  MoveL (T7763) to (103.84, 113.06, 9.7) mm, rotated rx 180 ry 0 rz -180 deg; joints [0, 0, 0, 0, 0, 0]
  Call Extruder 0.34896
  MoveL (T7764) to (111.94, 121.16, 9.7) mm, rotated rx 180 ry 0 rz -180 deg; joints [0, 0, 0, 0, 0, 0]
  Call Extruder 0.03385
  MoveL (T7765) to (113.06, 121.16, 9.7) mm, rotated rx 180 ry 0 rz -180 deg; joints [0, 0, 0, 0, 0, 0]
  Call Extruder 0.26282
  MoveL (T7766) to (119.16, 115.06, 9.7) mm, rotated rx 180 ry 0 rz -180 deg; joints [0, 0, 0, 0, 0, 0]
  Call Extruder 0.00278
  MoveL (T7767) to (119.09, 114.99, 9.7) mm, rotated rx 180 ry 0 rz -180 deg; joints [0, 0, 0, 0, 0, 0]
  Call Extruder 0.01541
  MoveL (T7768) to (119.09, 114.48, 9.7) mm, rotated rx 180 ry 0 rz -180 deg; joints [0, 0, 0, 0, 0, 0]
  Call Extruder 0.37671
  MoveL (T7769) to (110.35, 105.74, 9.7) mm, rotated rx 180 ry 0 rz -180 deg; joints [0, 0, 0, 0, 0, 0]
  Call Extruder 0.00909
  MoveL (T7770) to (110.05, 105.74, 9.7) mm, rotated rx 180 ry 0 rz -180 deg; joints [0, 0, 0, 0, 0, 0]
  Call Extruder 0.26727
  MoveL (T7771) to (103.84, 111.94, 9.7) mm, rotated rx 180 ry 0 rz -180 deg; joints [0, 0, 0, 0, 0, 0]
  Call Extruder 0.07441
  MoveL (T7772) to (103.84, 109.5, 9.7) mm, rotated rx 180 ry 0 rz -180 deg; joints [0, 0, 0, 0, 0, 0]
  Set speed (45.0 mm/s)
  Call Extruder -1.6
  MoveL (T7773) to (103.84, 109.5, 9.7) mm, rotated rx 180 ry 0 rz -180 deg; joints [0, 0, 0, 0, 0, 0]
  Set speed (120.0 mm/s)
  MoveL (T7774) to (103.84, 109.5, 9.7) mm, rotated rx 180 ry 0 rz -180 deg; joints [0, 0, 0, 0, 0, 0]
  Call Extruder -0.38
  MoveL (T7775) to (103.84, 110.57, 9.7) mm, rotated rx 180 ry 0 rz -180 deg; joints [0, 0, 0, 0, 0, 0]
  Set speed (45.0 mm/s)
  Call Extruder -0.02
  MoveL (T7776) to (103.84, 110.57, 9.7) mm, rotated rx 180 ry 0 rz -180 deg; joints [0, 0, 0, 0, 0, 0]
  Set speed (150.0 mm/s)
  MoveL (T7777) to (103.84, 110.57, 11.7) mm, rotated rx 180 ry 0 rz -180 deg; joints [0, 0, 0, 0, 0, 0]
  MoveL (T7778) to (104.34, 103.54, 11.7) mm, rotated rx 180 ry 0 rz -180 deg; joints [0, 0, 0, 0, 0, 0]
  MoveL (T7779) to (104.34, 103.54, 9.9) mm, rotated rx 180 ry 0 rz -180 deg; joints [0, 0, 0, 0, 0, 0]
  Set speed (40.0 mm/s)
  Call Extruder 2.0
  MoveL (T7780) to (104.34, 103.54, 9.9) mm, rotated rx 180 ry 0 rz -180 deg; joints [0, 0, 0, 0, 0, 0]
  Set speed (26.4 mm/s)
  MoveL (T7781) to (104.34, 103.54, 9.9) mm, rotated rx 180 ry 0 rz -180 deg; joints [0, 0, 0, 0, 0, 0]
  Call Extruder 0.16936
  MoveL (T7782) to (109.9, 103.54, 9.9) mm, rotated rx 180 ry 0 rz -180 deg; joints [0, 0, 0, 0, 0, 0]
  Call Extruder 0.05777
  MoveL (T7783) to (109.9, 105.44, 9.9) mm, rotated rx 180 ry 0 rz -180 deg; joints [0, 0, 0, 0, 0, 0]
  Call Extruder 0.12448
  MoveL (T7784) to (113.98, 105.44, 9.9) mm, rotated rx 180 ry 0 rz -180 deg; joints [0, 0, 0, 0, 0, 0]
  Call Extruder 0.05777
  MoveL (T7785) to (113.99, 103.54, 9.9) mm, rotated rx 180 ry 0 rz -180 deg; joints [0, 0, 0, 0, 0, 0]
  Call Extruder 0.2277
  MoveL (T7786) to (121.46, 103.54, 9.9) mm, rotated rx 180 ry 0 rz -180 deg; joints [0, 0, 0, 0, 0, 0]
  Call Extruder 0.19316
  MoveL (T7787) to (121.46, 109.88, 9.9) mm, rotated rx 180 ry 0 rz -180 deg; joints [0, 0, 0, 0, 0, 0]
  Call Extruder 0.05896
  MoveL (T7788) to (119.53, 109.88, 9.9) mm, rotated rx 180 ry 0 rz -180 deg; joints [0, 0, 0, 0, 0, 0]
  Call Extruder 0.13491
  MoveL (T7789) to (119.52, 114.31, 9.9) mm, rotated rx 180 ry 0 rz -180 deg; joints [0, 0, 0, 0, 0, 0]
  Call Extruder 0.05902
  MoveL (T7790) to (121.46, 114.31, 9.9) mm, rotated rx 180 ry 0 rz -180 deg; joints [0, 0, 0, 0, 0, 0]
  Call Extruder 0.21779
  MoveL (T7791) to (121.46, 121.46, 9.9) mm, rotated rx 180 ry 0 rz -180 deg; joints [0, 0, 0, 0, 0, 0]
  Call Extruder 0.54596
  MoveL (T7792) to (103.54, 121.46, 9.9) mm, rotated rx 180 ry 0 rz -180 deg; joints [0, 0, 0, 0, 0, 0]
  Call Extruder 0.54596
  MoveL (T7793) to (103.54, 103.54, 9.9) mm, rotated rx 180 ry 0 rz -180 deg; joints [0, 0, 0, 0, 0, 0]
  Call Extruder 0.02254
  MoveL (T7794) to (104.28, 103.54, 9.9) mm, rotated rx 180 ry 0 rz -180 deg; joints [0, 0, 0, 0, 0, 0]
  Set speed (150.0 mm/s)
  MoveL (T7795) to (103.53, 103.13, 9.9) mm, rotated rx 180 ry 0 rz -180 deg; joints [0, 0, 0, 0, 0, 0]
  Set speed (26.4 mm/s)
  MoveL (T7796) to (103.53, 103.13, 9.9) mm, rotated rx 180 ry 0 rz -180 deg; joints [0, 0, 0, 0, 0, 0]
  Call Extruder 0.20634
  MoveL (T7797) to (110.31, 103.13, 9.9) mm, rotated rx 180 ry 0 rz -180 deg; joints [0, 0, 0, 0, 0, 0]
  Call Extruder 0.05777
  MoveL (T7798) to (110.31, 105.03, 9.9) mm, rotated rx 180 ry 0 rz -180 deg; joints [0, 0, 0, 0, 0, 0]
  Call Extruder 0.09969
  MoveL (T7799) to (113.58, 105.03, 9.9) mm, rotated rx 180 ry 0 rz -180 deg; joints [0, 0, 0, 0, 0, 0]
  Call Extruder 0.05777
  MoveL (T7800) to (113.58, 103.13, 9.9) mm, rotated rx 180 ry 0 rz -180 deg; joints [0, 0, 0, 0, 0, 0]
  Call Extruder 0.2525
  MoveL (T7801) to (121.87, 103.13, 9.9) mm, rotated rx 180 ry 0 rz -180 deg; joints [0, 0, 0, 0, 0, 0]
  Call Extruder 0.21796
  MoveL (T7802) to (121.87, 110.29, 9.9) mm, rotated rx 180 ry 0 rz -180 deg; joints [0, 0, 0, 0, 0, 0]
  Call Extruder 0.05897
  MoveL (T7803) to (119.93, 110.29, 9.9) mm, rotated rx 180 ry 0 rz -180 deg; joints [0, 0, 0, 0, 0, 0]
  Call Extruder 0.11013
  MoveL (T7804) to (119.93, 113.9, 9.9) mm, rotated rx 180 ry 0 rz -180 deg; joints [0, 0, 0, 0, 0, 0]
  Call Extruder 0.05902
  MoveL (T7805) to (121.87, 113.91, 9.9) mm, rotated rx 180 ry 0 rz -180 deg; joints [0, 0, 0, 0, 0, 0]
  Call Extruder 0.24258
  MoveL (T7806) to (121.87, 121.87, 9.9) mm, rotated rx 180 ry 0 rz -180 deg; joints [0, 0, 0, 0, 0, 0]
  Call Extruder 0.57077
  MoveL (T7807) to (103.13, 121.87, 9.9) mm, rotated rx 180 ry 0 rz -180 deg; joints [0, 0, 0, 0, 0, 0]
  Call Extruder 0.57077
  MoveL (T7808) to (103.13, 103.13, 9.9) mm, rotated rx 180 ry 0 rz -180 deg; joints [0, 0, 0, 0, 0, 0]
  Call Extruder 0.01036
  MoveL (T7809) to (103.47, 103.13, 9.9) mm, rotated rx 180 ry 0 rz -180 deg; joints [0, 0, 0, 0, 0, 0]
  Set speed (150.0 mm/s)
  MoveL (T7810) to (102.72, 102.81, 9.9) mm, rotated rx 180 ry 0 rz -180 deg; joints [0, 0, 0, 0, 0, 0]
  Set speed (25.0 mm/s)
  MoveL (T7811) to (102.72, 102.81, 9.9) mm, rotated rx 180 ry 0 rz -180 deg; joints [0, 0, 0, 0, 0, 0]
  Call Extruder 0.00259
  MoveL (T7812) to (102.72, 102.72, 9.9) mm, rotated rx 180 ry 0 rz -180 deg; joints [0, 0, 0, 0, 0, 0]
  Call Extruder 0.24332
  MoveL (T7813) to (110.71, 102.72, 9.9) mm, rotated rx 180 ry 0 rz -180 deg; joints [0, 0, 0, 0, 0, 0]
  Call Extruder 0.05777
  MoveL (T7814) to (110.71, 104.62, 9.9) mm, rotated rx 180 ry 0 rz -180 deg; joints [0, 0, 0, 0, 0, 0]
  Call Extruder 0.0749
  MoveL (T7815) to (113.17, 104.62, 9.9) mm, rotated rx 180 ry 0 rz -180 deg; joints [0, 0, 0, 0, 0, 0]
  Call Extruder 0.05777
  MoveL (T7816) to (113.17, 102.72, 9.9) mm, rotated rx 180 ry 0 rz -180 deg; joints [0, 0, 0, 0, 0, 0]
  Call Extruder 0.27729
  MoveL (T7817) to (122.28, 102.72, 9.9) mm, rotated rx 180 ry 0 rz -180 deg; joints [0, 0, 0, 0, 0, 0]
  Call Extruder 0.24275
  MoveL (T7818) to (122.28, 110.69, 9.9) mm, rotated rx 180 ry 0 rz -180 deg; joints [0, 0, 0, 0, 0, 0]
  Call Extruder 0.05897
  MoveL (T7819) to (120.34, 110.69, 9.9) mm, rotated rx 180 ry 0 rz -180 deg; joints [0, 0, 0, 0, 0, 0]
  Call Extruder 0.08535
  MoveL (T7820) to (120.34, 113.5, 9.9) mm, rotated rx 180 ry 0 rz -180 deg; joints [0, 0, 0, 0, 0, 0]
  Call Extruder 0.05901
  MoveL (T7821) to (122.28, 113.5, 9.9) mm, rotated rx 180 ry 0 rz -180 deg; joints [0, 0, 0, 0, 0, 0]
  Call Extruder 0.26736
  MoveL (T7822) to (122.28, 122.28, 9.9) mm, rotated rx 180 ry 0 rz -180 deg; joints [0, 0, 0, 0, 0, 0]
  Call Extruder 0.59557
  MoveL (T7823) to (102.72, 122.28, 9.9) mm, rotated rx 180 ry 0 rz -180 deg; joints [0, 0, 0, 0, 0, 0]
  Call Extruder 0.59115
  MoveL (T7824) to (102.72, 102.87, 9.9) mm, rotated rx 180 ry 0 rz -180 deg; joints [0, 0, 0, 0, 0, 0]
  Set speed (150.0 mm/s)
  MoveL (T7825) to (102.78, 102.75, 9.9) mm, rotated rx 180 ry 0 rz -180 deg; joints [0, 0, 0, 0, 0, 0]
  Set speed (45.0 mm/s)
  Call Extruder -1.6
  MoveL (T7826) to (102.78, 102.75, 9.9) mm, rotated rx 180 ry 0 rz -180 deg; joints [0, 0, 0, 0, 0, 0]
  Set speed (120.0 mm/s)
  MoveL (T7827) to (102.78, 102.75, 9.9) mm, rotated rx 180 ry 0 rz -180 deg; joints [0, 0, 0, 0, 0, 0]
  Call Extruder -0.05166
  MoveL (T7828) to (102.72, 102.72, 9.9) mm, rotated rx 180 ry 0 rz -180 deg; joints [0, 0, 0, 0, 0, 0]
  Call Extruder -0.32834
  MoveL (T7829) to (103.65, 102.72, 9.9) mm, rotated rx 180 ry 0 rz -180 deg; joints [0, 0, 0, 0, 0, 0]
  Set speed (45.0 mm/s)
  Call Extruder -0.02
  MoveL (T7830) to (103.65, 102.72, 9.9) mm, rotated rx 180 ry 0 rz -180 deg; joints [0, 0, 0, 0, 0, 0]
  Set speed (150.0 mm/s)
  MoveL (T7831) to (103.65, 102.72, 11.9) mm, rotated rx 180 ry 0 rz -180 deg; joints [0, 0, 0, 0, 0, 0]
  MoveL (T7832) to (106.29, 103.84, 11.9) mm, rotated rx 180 ry 0 rz -180 deg; joints [0, 0, 0, 0, 0, 0]
  MoveL (T7833) to (106.29, 103.84, 9.9) mm, rotated rx 180 ry 0 rz -180 deg; joints [0, 0, 0, 0, 0, 0]
  Set speed (40.0 mm/s)
  Call Extruder 2.0
  MoveL (T7834) to (106.29, 103.84, 9.9) mm, rotated rx 180 ry 0 rz -180 deg; joints [0, 0, 0, 0, 0, 0]
  Set speed (26.4 mm/s)
  MoveL (T7835) to (106.29, 103.84, 9.9) mm, rotated rx 180 ry 0 rz -180 deg; joints [0, 0, 0, 0, 0, 0]
  Call Extruder 0.07441
  MoveL (T7836) to (103.84, 103.84, 9.9) mm, rotated rx 180 ry 0 rz -180 deg; joints [0, 0, 0, 0, 0, 0]
  Call Extruder 0.7458
  MoveL (T7837) to (121.16, 121.16, 9.9) mm, rotated rx 180 ry 0 rz -180 deg; joints [0, 0, 0, 0, 0, 0]
  Call Extruder 0.07441
  MoveL (T7838) to (118.71, 121.16, 9.9) mm, rotated rx 180 ry 0 rz -180 deg; joints [0, 0, 0, 0, 0, 0]
  Set speed (45.0 mm/s)
  Call Extruder -1.6
  MoveL (T7839) to (118.71, 121.16, 9.9) mm, rotated rx 180 ry 0 rz -180 deg; joints [0, 0, 0, 0, 0, 0]
  Set speed (120.0 mm/s)
  MoveL (T7840) to (118.71, 121.16, 9.9) mm, rotated rx 180 ry 0 rz -180 deg; joints [0, 0, 0, 0, 0, 0]
  Call Extruder -0.38
  MoveL (T7841) to (119.78, 121.16, 9.9) mm, rotated rx 180 ry 0 rz -180 deg; joints [0, 0, 0, 0, 0, 0]
  Set speed (45.0 mm/s)
  Call Extruder -0.02
  MoveL (T7842) to (119.78, 121.16, 9.9) mm, rotated rx 180 ry 0 rz -180 deg; joints [0, 0, 0, 0, 0, 0]
  Set speed (150.0 mm/s)
  MoveL (T7843) to (119.78, 121.16, 11.9) mm, rotated rx 180 ry 0 rz -180 deg; joints [0, 0, 0, 0, 0, 0]
  MoveL (T7844) to (121.16, 116.35, 11.9) mm, rotated rx 180 ry 0 rz -180 deg; joints [0, 0, 0, 0, 0, 0]
  MoveL (T7845) to (121.16, 116.35, 9.9) mm, rotated rx 180 ry 0 rz -180 deg; joints [0, 0, 0, 0, 0, 0]
  Set speed (40.0 mm/s)
  Call Extruder 2.0
  MoveL (T7846) to (121.16, 116.35, 9.9) mm, rotated rx 180 ry 0 rz -180 deg; joints [0, 0, 0, 0, 0, 0]
  Set speed (26.4 mm/s)
  MoveL (T7847) to (121.16, 116.35, 9.9) mm, rotated rx 180 ry 0 rz -180 deg; joints [0, 0, 0, 0, 0, 0]
  Call Extruder 0.02808
  MoveL (T7848) to (121.16, 115.42, 9.9) mm, rotated rx 180 ry 0 rz -180 deg; joints [0, 0, 0, 0, 0, 0]
  Call Extruder 0.03432
  MoveL (T7849) to (120.03, 115.42, 9.9) mm, rotated rx 180 ry 0 rz -180 deg; joints [0, 0, 0, 0, 0, 0]
  Call Extruder 0.04854
  MoveL (T7850) to (121.16, 116.55, 9.9) mm, rotated rx 180 ry 0 rz -180 deg; joints [0, 0, 0, 0, 0, 0]
  Call Extruder 0.03385
  MoveL (T7851) to (121.16, 117.66, 9.9) mm, rotated rx 180 ry 0 rz -180 deg; joints [0, 0, 0, 0, 0, 0]
  Call Extruder 0.15054
  MoveL (T7852) to (117.66, 121.16, 9.9) mm, rotated rx 180 ry 0 rz -180 deg; joints [0, 0, 0, 0, 0, 0]
  Call Extruder 0.03385
  MoveL (T7853) to (116.55, 121.16, 9.9) mm, rotated rx 180 ry 0 rz -180 deg; joints [0, 0, 0, 0, 0, 0]
  Call Extruder 0.54738
  MoveL (T7854) to (103.84, 108.45, 9.9) mm, rotated rx 180 ry 0 rz -180 deg; joints [0, 0, 0, 0, 0, 0]
  Call Extruder 0.03385
  MoveL (T7855) to (103.84, 107.34, 9.9) mm, rotated rx 180 ry 0 rz -180 deg; joints [0, 0, 0, 0, 0, 0]
  Call Extruder 0.15054
  MoveL (T7856) to (107.34, 103.84, 9.9) mm, rotated rx 180 ry 0 rz -180 deg; joints [0, 0, 0, 0, 0, 0]
  Call Extruder 0.03385
  MoveL (T7857) to (108.45, 103.84, 9.9) mm, rotated rx 180 ry 0 rz -180 deg; joints [0, 0, 0, 0, 0, 0]
  Call Extruder 0.02461
  MoveL (T7858) to (109.02, 104.42, 9.9) mm, rotated rx 180 ry 0 rz -180 deg; joints [0, 0, 0, 0, 0, 0]
  Call Extruder 0.03458
  MoveL (T7859) to (109.02, 105.55, 9.9) mm, rotated rx 180 ry 0 rz -180 deg; joints [0, 0, 0, 0, 0, 0]
  Call Extruder 0.01376
  MoveL (T7860) to (109.34, 105.87, 9.9) mm, rotated rx 180 ry 0 rz -180 deg; joints [0, 0, 0, 0, 0, 0]
  Call Extruder 0.01427
  MoveL (T7861) to (109.81, 105.87, 9.9) mm, rotated rx 180 ry 0 rz -180 deg; joints [0, 0, 0, 0, 0, 0]
  Call Extruder 0.00269
  MoveL (T7862) to (109.87, 105.81, 9.9) mm, rotated rx 180 ry 0 rz -180 deg; joints [0, 0, 0, 0, 0, 0]
  Set speed (150.0 mm/s)
  MoveL (T7863) to (109.78, 104.52, 9.9) mm, rotated rx 180 ry 0 rz -180 deg; joints [0, 0, 0, 0, 0, 0]
  Set speed (26.4 mm/s)
  MoveL (T7864) to (109.78, 104.52, 9.9) mm, rotated rx 180 ry 0 rz -180 deg; joints [0, 0, 0, 0, 0, 0]
  Call Extruder 0.01563
  MoveL (T7865) to (109.43, 104.17, 9.9) mm, rotated rx 180 ry 0 rz -180 deg; joints [0, 0, 0, 0, 0, 0]
  Call Extruder 0.01901
  MoveL (T7866) to (109.43, 104.77, 9.9) mm, rotated rx 180 ry 0 rz -180 deg; joints [0, 0, 0, 0, 0, 0]
  Call Extruder 0.00741
  MoveL (T7867) to (109.59, 104.94, 9.9) mm, rotated rx 180 ry 0 rz -180 deg; joints [0, 0, 0, 0, 0, 0]
  Call Extruder 0.01671
  MoveL (T7868) to (109.59, 105.46, 9.9) mm, rotated rx 180 ry 0 rz -180 deg; joints [0, 0, 0, 0, 0, 0]
  Call Extruder 0.0023
  MoveL (T7869) to (109.52, 105.46, 9.9) mm, rotated rx 180 ry 0 rz -180 deg; joints [0, 0, 0, 0, 0, 0]
  Call Extruder 0.01238
  MoveL (T7870) to (109.25, 105.19, 9.9) mm, rotated rx 180 ry 0 rz -180 deg; joints [0, 0, 0, 0, 0, 0]
  Set speed (45.0 mm/s)
  Call Extruder -1.6
  MoveL (T7871) to (109.25, 105.19, 9.9) mm, rotated rx 180 ry 0 rz -180 deg; joints [0, 0, 0, 0, 0, 0]
  Set speed (120.0 mm/s)
  MoveL (T7872) to (109.25, 105.19, 9.9) mm, rotated rx 180 ry 0 rz -180 deg; joints [0, 0, 0, 0, 0, 0]
  Call Extruder -0.13905
  MoveL (T7873) to (109.52, 105.46, 9.9) mm, rotated rx 180 ry 0 rz -180 deg; joints [0, 0, 0, 0, 0, 0]
  Call Extruder -0.02586
  MoveL (T7874) to (109.59, 105.46, 9.9) mm, rotated rx 180 ry 0 rz -180 deg; joints [0, 0, 0, 0, 0, 0]
  Call Extruder -0.18771
  MoveL (T7875) to (109.59, 104.94, 9.9) mm, rotated rx 180 ry 0 rz -180 deg; joints [0, 0, 0, 0, 0, 0]
  Call Extruder -0.02738
  MoveL (T7876) to (109.54, 104.88, 9.9) mm, rotated rx 180 ry 0 rz -180 deg; joints [0, 0, 0, 0, 0, 0]
  Set speed (45.0 mm/s)
  Call Extruder -0.02
  MoveL (T7877) to (109.54, 104.88, 9.9) mm, rotated rx 180 ry 0 rz -180 deg; joints [0, 0, 0, 0, 0, 0]
  Set speed (150.0 mm/s)
  MoveL (T7878) to (109.54, 104.88, 11.9) mm, rotated rx 180 ry 0 rz -180 deg; joints [0, 0, 0, 0, 0, 0]
  MoveL (T7879) to (112.14, 105.74, 11.9) mm, rotated rx 180 ry 0 rz -180 deg; joints [0, 0, 0, 0, 0, 0]
  MoveL (T7880) to (112.14, 105.74, 9.9) mm, rotated rx 180 ry 0 rz -180 deg; joints [0, 0, 0, 0, 0, 0]
  Set speed (40.0 mm/s)
  Call Extruder 2.0
  MoveL (T7881) to (112.14, 105.74, 9.9) mm, rotated rx 180 ry 0 rz -180 deg; joints [0, 0, 0, 0, 0, 0]
  Set speed (26.4 mm/s)
  MoveL (T7882) to (112.14, 105.74, 9.9) mm, rotated rx 180 ry 0 rz -180 deg; joints [0, 0, 0, 0, 0, 0]
  Call Extruder 0.05515
  MoveL (T7883) to (113.95, 105.74, 9.9) mm, rotated rx 180 ry 0 rz -180 deg; joints [0, 0, 0, 0, 0, 0]
  Call Extruder 0.00557
  MoveL (T7884) to (114.08, 105.87, 9.9) mm, rotated rx 180 ry 0 rz -180 deg; joints [0, 0, 0, 0, 0, 0]
  Call Extruder 0.01369
  MoveL (T7885) to (114.52, 105.87, 9.9) mm, rotated rx 180 ry 0 rz -180 deg; joints [0, 0, 0, 0, 0, 0]
  Call Extruder 0.46011
  MoveL (T7886) to (103.84, 116.55, 9.9) mm, rotated rx 180 ry 0 rz -180 deg; joints [0, 0, 0, 0, 0, 0]
  Call Extruder 0.03385
  MoveL (T7887) to (103.84, 117.66, 9.9) mm, rotated rx 180 ry 0 rz -180 deg; joints [0, 0, 0, 0, 0, 0]
  Call Extruder 0.15054
  MoveL (T7888) to (107.34, 121.16, 9.9) mm, rotated rx 180 ry 0 rz -180 deg; joints [0, 0, 0, 0, 0, 0]
  Call Extruder 0.03385
  MoveL (T7889) to (108.45, 121.16, 9.9) mm, rotated rx 180 ry 0 rz -180 deg; joints [0, 0, 0, 0, 0, 0]
  Call Extruder 0.46399
  MoveL (T7890) to (119.22, 110.39, 9.9) mm, rotated rx 180 ry 0 rz -180 deg; joints [0, 0, 0, 0, 0, 0]
  Call Extruder 0.01148
  MoveL (T7891) to (119.22, 110.01, 9.9) mm, rotated rx 180 ry 0 rz -180 deg; joints [0, 0, 0, 0, 0, 0]
  Call Extruder 0.18856
  MoveL (T7892) to (114.84, 105.63, 9.9) mm, rotated rx 180 ry 0 rz -180 deg; joints [0, 0, 0, 0, 0, 0]
  Call Extruder 0.00351
  MoveL (T7893) to (114.92, 105.55, 9.9) mm, rotated rx 180 ry 0 rz -180 deg; joints [0, 0, 0, 0, 0, 0]
  Call Extruder 0.00247
  MoveL (T7894) to (114.92, 105.47, 9.9) mm, rotated rx 180 ry 0 rz -180 deg; joints [0, 0, 0, 0, 0, 0]
  Call Extruder 0.07002
  MoveL (T7895) to (116.55, 103.84, 9.9) mm, rotated rx 180 ry 0 rz -180 deg; joints [0, 0, 0, 0, 0, 0]
  Call Extruder 0.03385
  MoveL (T7896) to (117.66, 103.84, 9.9) mm, rotated rx 180 ry 0 rz -180 deg; joints [0, 0, 0, 0, 0, 0]
  Call Extruder 0.15054
  MoveL (T7897) to (121.16, 107.34, 9.9) mm, rotated rx 180 ry 0 rz -180 deg; joints [0, 0, 0, 0, 0, 0]
  Call Extruder 0.03385
  MoveL (T7898) to (121.16, 108.45, 9.9) mm, rotated rx 180 ry 0 rz -180 deg; joints [0, 0, 0, 0, 0, 0]
  Call Extruder 0.01201
  MoveL (T7899) to (120.88, 108.73, 9.9) mm, rotated rx 180 ry 0 rz -180 deg; joints [0, 0, 0, 0, 0, 0]
  Call Extruder 0.04458
  MoveL (T7900) to (119.41, 108.73, 9.9) mm, rotated rx 180 ry 0 rz -180 deg; joints [0, 0, 0, 0, 0, 0]
  Call Extruder 0.01373
  MoveL (T7901) to (119.09, 109.05, 9.9) mm, rotated rx 180 ry 0 rz -180 deg; joints [0, 0, 0, 0, 0, 0]
  Call Extruder 0.01609
  MoveL (T7902) to (119.09, 109.58, 9.9) mm, rotated rx 180 ry 0 rz -180 deg; joints [0, 0, 0, 0, 0, 0]
  Set speed (45.0 mm/s)
  Call Extruder -1.6
  MoveL (T7903) to (119.09, 109.58, 9.9) mm, rotated rx 180 ry 0 rz -180 deg; joints [0, 0, 0, 0, 0, 0]
  Set speed (120.0 mm/s)
  MoveL (T7904) to (119.09, 109.58, 9.9) mm, rotated rx 180 ry 0 rz -180 deg; joints [0, 0, 0, 0, 0, 0]
  Call Extruder -0.18818
  MoveL (T7905) to (119.09, 109.05, 9.9) mm, rotated rx 180 ry 0 rz -180 deg; joints [0, 0, 0, 0, 0, 0]
  Call Extruder -0.16059
  MoveL (T7906) to (119.41, 108.73, 9.9) mm, rotated rx 180 ry 0 rz -180 deg; joints [0, 0, 0, 0, 0, 0]
  Call Extruder -0.03122
  MoveL (T7907) to (119.5, 108.73, 9.9) mm, rotated rx 180 ry 0 rz -180 deg; joints [0, 0, 0, 0, 0, 0]
  Set speed (45.0 mm/s)
  Call Extruder -0.02
  MoveL (T7908) to (119.5, 108.73, 9.9) mm, rotated rx 180 ry 0 rz -180 deg; joints [0, 0, 0, 0, 0, 0]
  Set speed (150.0 mm/s)
  MoveL (T7909) to (119.5, 108.73, 11.9) mm, rotated rx 180 ry 0 rz -180 deg; joints [0, 0, 0, 0, 0, 0]
  MoveL (T7910) to (121.34, 109.33, 11.9) mm, rotated rx 180 ry 0 rz -180 deg; joints [0, 0, 0, 0, 0, 0]
  MoveL (T7911) to (121.34, 109.33, 9.9) mm, rotated rx 180 ry 0 rz -180 deg; joints [0, 0, 0, 0, 0, 0]
  Set speed (40.0 mm/s)
  Call Extruder 2.0
  MoveL (T7912) to (121.34, 109.33, 9.9) mm, rotated rx 180 ry 0 rz -180 deg; joints [0, 0, 0, 0, 0, 0]
  Set speed (26.4 mm/s)
  MoveL (T7913) to (121.34, 109.33, 9.9) mm, rotated rx 180 ry 0 rz -180 deg; joints [0, 0, 0, 0, 0, 0]
  Call Extruder 0.01001
  MoveL (T7914) to (121.14, 109.14, 9.9) mm, rotated rx 180 ry 0 rz -180 deg; joints [0, 0, 0, 0, 0, 0]
  Call Extruder 0.02524
  MoveL (T7915) to (120.45, 109.14, 9.9) mm, rotated rx 180 ry 0 rz -180 deg; joints [0, 0, 0, 0, 0, 0]
  Call Extruder 0.02268
  MoveL (T7916) to (120.89, 109.58, 9.9) mm, rotated rx 180 ry 0 rz -180 deg; joints [0, 0, 0, 0, 0, 0]
  Call Extruder 0.02524
  MoveL (T7917) to (120.2, 109.58, 9.9) mm, rotated rx 180 ry 0 rz -180 deg; joints [0, 0, 0, 0, 0, 0]
  Call Extruder 0.02268
  MoveL (T7918) to (119.76, 109.14, 9.9) mm, rotated rx 180 ry 0 rz -180 deg; joints [0, 0, 0, 0, 0, 0]
  Call Extruder 0.00667
  MoveL (T7919) to (119.58, 109.14, 9.9) mm, rotated rx 180 ry 0 rz -180 deg; joints [0, 0, 0, 0, 0, 0]
  Call Extruder 0.00418
  MoveL (T7920) to (119.5, 109.22, 9.9) mm, rotated rx 180 ry 0 rz -180 deg; joints [0, 0, 0, 0, 0, 0]
  Call Extruder 0.01263
  MoveL (T7921) to (119.5, 109.56, 9.9) mm, rotated rx 180 ry 0 rz -180 deg; joints [0, 0, 0, 0, 0, 0]
  Call Extruder 0.01011
  MoveL (T7922) to (119.69, 109.76, 9.9) mm, rotated rx 180 ry 0 rz -180 deg; joints [0, 0, 0, 0, 0, 0]
  Set speed (45.0 mm/s)
  Call Extruder -1.6
  MoveL (T7923) to (119.69, 109.76, 9.9) mm, rotated rx 180 ry 0 rz -180 deg; joints [0, 0, 0, 0, 0, 0]
  Set speed (120.0 mm/s)
  MoveL (T7924) to (119.69, 109.76, 9.9) mm, rotated rx 180 ry 0 rz -180 deg; joints [0, 0, 0, 0, 0, 0]
  Call Extruder -0.09855
  MoveL (T7925) to (119.5, 109.56, 9.9) mm, rotated rx 180 ry 0 rz -180 deg; joints [0, 0, 0, 0, 0, 0]
  Call Extruder -0.1231
  MoveL (T7926) to (119.5, 109.22, 9.9) mm, rotated rx 180 ry 0 rz -180 deg; joints [0, 0, 0, 0, 0, 0]
  Call Extruder -0.04075
  MoveL (T7927) to (119.58, 109.14, 9.9) mm, rotated rx 180 ry 0 rz -180 deg; joints [0, 0, 0, 0, 0, 0]
  Call Extruder -0.06497
  MoveL (T7928) to (119.76, 109.14, 9.9) mm, rotated rx 180 ry 0 rz -180 deg; joints [0, 0, 0, 0, 0, 0]
  Call Extruder -0.05262
  MoveL (T7929) to (119.87, 109.24, 9.9) mm, rotated rx 180 ry 0 rz -180 deg; joints [0, 0, 0, 0, 0, 0]
  Set speed (45.0 mm/s)
  Call Extruder -0.02
  MoveL (T7930) to (119.87, 109.24, 9.9) mm, rotated rx 180 ry 0 rz -180 deg; joints [0, 0, 0, 0, 0, 0]
  Set speed (150.0 mm/s)
  MoveL (T7931) to (119.87, 109.24, 11.9) mm, rotated rx 180 ry 0 rz -180 deg; joints [0, 0, 0, 0, 0, 0]
  MoveL (T7932) to (121.14, 115.2, 11.9) mm, rotated rx 180 ry 0 rz -180 deg; joints [0, 0, 0, 0, 0, 0]
  MoveL (T7933) to (121.14, 115.2, 9.9) mm, rotated rx 180 ry 0 rz -180 deg; joints [0, 0, 0, 0, 0, 0]
  Set speed (40.0 mm/s)
  Call Extruder 2.0
  MoveL (T7934) to (121.14, 115.2, 9.9) mm, rotated rx 180 ry 0 rz -180 deg; joints [0, 0, 0, 0, 0, 0]
  Set speed (26.4 mm/s)
  MoveL (T7935) to (121.14, 115.2, 9.9) mm, rotated rx 180 ry 0 rz -180 deg; joints [0, 0, 0, 0, 0, 0]
  Call Extruder 0.02922
  MoveL (T7936) to (120.56, 114.62, 9.9) mm, rotated rx 180 ry 0 rz -180 deg; joints [0, 0, 0, 0, 0, 0]
  Call Extruder 0.02361
  MoveL (T7937) to (119.89, 114.61, 9.9) mm, rotated rx 180 ry 0 rz -180 deg; joints [0, 0, 0, 0, 0, 0]
  Call Extruder 0.02006
  MoveL (T7938) to (120.29, 115.02, 9.9) mm, rotated rx 180 ry 0 rz -180 deg; joints [0, 0, 0, 0, 0, 0]
  Call Extruder 0.02361
  MoveL (T7939) to (119.62, 115.02, 9.9) mm, rotated rx 180 ry 0 rz -180 deg; joints [0, 0, 0, 0, 0, 0]
  Call Extruder 0.0155
  MoveL (T7940) to (119.31, 114.7, 9.9) mm, rotated rx 180 ry 0 rz -180 deg; joints [0, 0, 0, 0, 0, 0]
  Set speed (45.0 mm/s)
  Call Extruder -1.6
  MoveL (T7941) to (119.31, 114.7, 9.9) mm, rotated rx 180 ry 0 rz -180 deg; joints [0, 0, 0, 0, 0, 0]
  Set speed (120.0 mm/s)
  MoveL (T7942) to (119.31, 114.7, 9.9) mm, rotated rx 180 ry 0 rz -180 deg; joints [0, 0, 0, 0, 0, 0]
  Call Extruder -0.15638
  MoveL (T7943) to (119.62, 115.02, 9.9) mm, rotated rx 180 ry 0 rz -180 deg; joints [0, 0, 0, 0, 0, 0]
  Call Extruder -0.22362
  MoveL (T7944) to (120.25, 115.02, 9.9) mm, rotated rx 180 ry 0 rz -180 deg; joints [0, 0, 0, 0, 0, 0]
  Set speed (45.0 mm/s)
  Call Extruder -0.02
  MoveL (T7945) to (120.25, 115.02, 9.9) mm, rotated rx 180 ry 0 rz -180 deg; joints [0, 0, 0, 0, 0, 0]
  Set speed (150.0 mm/s)
  MoveL (T7946) to (120.25, 115.02, 11.9) mm, rotated rx 180 ry 0 rz -180 deg; joints [0, 0, 0, 0, 0, 0]
  MoveL (T7947) to (118.71, 103.84, 11.9) mm, rotated rx 180 ry 0 rz -180 deg; joints [0, 0, 0, 0, 0, 0]
  MoveL (T7948) to (118.71, 103.84, 9.9) mm, rotated rx 180 ry 0 rz -180 deg; joints [0, 0, 0, 0, 0, 0]
  Set speed (40.0 mm/s)
  Call Extruder 2.0
  MoveL (T7949) to (118.71, 103.84, 9.9) mm, rotated rx 180 ry 0 rz -180 deg; joints [0, 0, 0, 0, 0, 0]
  Set speed (26.4 mm/s)
  MoveL (T7950) to (118.71, 103.84, 9.9) mm, rotated rx 180 ry 0 rz -180 deg; joints [0, 0, 0, 0, 0, 0]
  Call Extruder 0.07441
  MoveL (T7951) to (121.16, 103.84, 9.9) mm, rotated rx 180 ry 0 rz -180 deg; joints [0, 0, 0, 0, 0, 0]
  Call Extruder 0.7458
  MoveL (T7952) to (103.84, 121.16, 9.9) mm, rotated rx 180 ry 0 rz -180 deg; joints [0, 0, 0, 0, 0, 0]
  Call Extruder 0.07441
  MoveL (T7953) to (106.29, 121.16, 9.9) mm, rotated rx 180 ry 0 rz -180 deg; joints [0, 0, 0, 0, 0, 0]
  Set speed (45.0 mm/s)
  Call Extruder -1.6
  MoveL (T7954) to (106.29, 121.16, 9.9) mm, rotated rx 180 ry 0 rz -180 deg; joints [0, 0, 0, 0, 0, 0]
  Set speed (120.0 mm/s)
  MoveL (T7955) to (106.29, 121.16, 9.9) mm, rotated rx 180 ry 0 rz -180 deg; joints [0, 0, 0, 0, 0, 0]
  Call Extruder -0.38
  MoveL (T7956) to (105.22, 121.16, 9.9) mm, rotated rx 180 ry 0 rz -180 deg; joints [0, 0, 0, 0, 0, 0]
  Set speed (45.0 mm/s)
  Call Extruder -0.02
  MoveL (T7957) to (105.22, 121.16, 9.9) mm, rotated rx 180 ry 0 rz -180 deg; joints [0, 0, 0, 0, 0, 0]
  Set speed (150.0 mm/s)
  MoveL (T7958) to (105.22, 121.16, 11.9) mm, rotated rx 180 ry 0 rz -180 deg; joints [0, 0, 0, 0, 0, 0]
  MoveL (T7959) to (103.84, 115.5, 11.9) mm, rotated rx 180 ry 0 rz -180 deg; joints [0, 0, 0, 0, 0, 0]
  MoveL (T7960) to (103.84, 115.5, 9.9) mm, rotated rx 180 ry 0 rz -180 deg; joints [0, 0, 0, 0, 0, 0]
  Set speed (40.0 mm/s)
  Call Extruder 2.0
  MoveL (T7961) to (103.84, 115.5, 9.9) mm, rotated rx 180 ry 0 rz -180 deg; joints [0, 0, 0, 0, 0, 0]
  Set speed (26.4 mm/s)
  MoveL (T7962) to (103.84, 115.5, 9.9) mm, rotated rx 180 ry 0 rz -180 deg; joints [0, 0, 0, 0, 0, 0]
  Call Extruder 0.07441
  MoveL (T7963) to (103.84, 113.06, 9.9) mm, rotated rx 180 ry 0 rz -180 deg; joints [0, 0, 0, 0, 0, 0]
  Call Extruder 0.34896
  MoveL (T7964) to (111.94, 121.16, 9.9) mm, rotated rx 180 ry 0 rz -180 deg; joints [0, 0, 0, 0, 0, 0]
  Call Extruder 0.03385
  MoveL (T7965) to (113.06, 121.16, 9.9) mm, rotated rx 180 ry 0 rz -180 deg; joints [0, 0, 0, 0, 0, 0]
  Call Extruder 0.26038
  MoveL (T7966) to (119.1, 115.11, 9.9) mm, rotated rx 180 ry 0 rz -180 deg; joints [0, 0, 0, 0, 0, 0]
  Call Extruder 0.0191
  MoveL (T7967) to (119.09, 114.48, 9.9) mm, rotated rx 180 ry 0 rz -180 deg; joints [0, 0, 0, 0, 0, 0]
  Call Extruder 0.37671
  MoveL (T7968) to (110.35, 105.74, 9.9) mm, rotated rx 180 ry 0 rz -180 deg; joints [0, 0, 0, 0, 0, 0]
  Call Extruder 0.0091
  MoveL (T7969) to (110.05, 105.74, 9.9) mm, rotated rx 180 ry 0 rz -180 deg; joints [0, 0, 0, 0, 0, 0]
  Call Extruder 0.26726
  MoveL (T7970) to (103.84, 111.94, 9.9) mm, rotated rx 180 ry 0 rz -180 deg; joints [0, 0, 0, 0, 0, 0]
  Call Extruder 0.07441
  MoveL (T7971) to (103.84, 109.5, 9.9) mm, rotated rx 180 ry 0 rz -180 deg; joints [0, 0, 0, 0, 0, 0]
  Set speed (45.0 mm/s)
  Call Extruder -1.6
  MoveL (T7972) to (103.84, 109.5, 9.9) mm, rotated rx 180 ry 0 rz -180 deg; joints [0, 0, 0, 0, 0, 0]
  Set speed (120.0 mm/s)
  MoveL (T7973) to (103.84, 109.5, 9.9) mm, rotated rx 180 ry 0 rz -180 deg; joints [0, 0, 0, 0, 0, 0]
  Call Extruder -0.38
  MoveL (T7974) to (103.84, 110.57, 9.9) mm, rotated rx 180 ry 0 rz -180 deg; joints [0, 0, 0, 0, 0, 0]
  Set speed (45.0 mm/s)
  Call Extruder -0.02
  MoveL (T7975) to (103.84, 110.57, 9.9) mm, rotated rx 180 ry 0 rz -180 deg; joints [0, 0, 0, 0, 0, 0]
  Set speed (150.0 mm/s)
  MoveL (T7976) to (103.84, 110.57, 11.9) mm, rotated rx 180 ry 0 rz -180 deg; joints [0, 0, 0, 0, 0, 0]
  MoveL (T7977) to (114.11, 104.04, 11.9) mm, rotated rx 180 ry 0 rz -180 deg; joints [0, 0, 0, 0, 0, 0]
  MoveL (T7978) to (114.11, 104.04, 9.9) mm, rotated rx 180 ry 0 rz -180 deg; joints [0, 0, 0, 0, 0, 0]
  Set speed (40.0 mm/s)
  Call Extruder 2.0
  MoveL (T7979) to (114.11, 104.04, 9.9) mm, rotated rx 180 ry 0 rz -180 deg; joints [0, 0, 0, 0, 0, 0]
  Set speed (26.4 mm/s)
  MoveL (T7980) to (114.11, 104.04, 9.9) mm, rotated rx 180 ry 0 rz -180 deg; joints [0, 0, 0, 0, 0, 0]
  Call Extruder 0.0193
  MoveL (T7981) to (114.52, 104.45, 9.9) mm, rotated rx 180 ry 0 rz -180 deg; joints [0, 0, 0, 0, 0, 0]
  Call Extruder 0.02093
  MoveL (T7982) to (114.52, 105.08, 9.9) mm, rotated rx 180 ry 0 rz -180 deg; joints [0, 0, 0, 0, 0, 0]
  Call Extruder 0.0193
  MoveL (T7983) to (114.11, 104.67, 9.9) mm, rotated rx 180 ry 0 rz -180 deg; joints [0, 0, 0, 0, 0, 0]
  Set speed (45.0 mm/s)
  Call Extruder -1.6
  MoveL (T7984) to (114.11, 104.67, 9.9) mm, rotated rx 180 ry 0 rz -180 deg; joints [0, 0, 0, 0, 0, 0]
  Set speed (120.0 mm/s)
  MoveL (T7985) to (114.11, 104.67, 9.9) mm, rotated rx 180 ry 0 rz -180 deg; joints [0, 0, 0, 0, 0, 0]
  Call Extruder -0.20654
  MoveL (T7986) to (114.52, 105.08, 9.9) mm, rotated rx 180 ry 0 rz -180 deg; joints [0, 0, 0, 0, 0, 0]
  Call Extruder -0.17346
  MoveL (T7987) to (114.52, 104.59, 9.9) mm, rotated rx 180 ry 0 rz -180 deg; joints [0, 0, 0, 0, 0, 0]
  Set speed (45.0 mm/s)
  Call Extruder -0.02
  MoveL (T7988) to (114.52, 104.59, 9.9) mm, rotated rx 180 ry 0 rz -180 deg; joints [0, 0, 0, 0, 0, 0]
  Set speed (150.0 mm/s)
  MoveL (T7989) to (114.52, 104.59, 11.9) mm, rotated rx 180 ry 0 rz -180 deg; joints [0, 0, 0, 0, 0, 0]
  MoveL (T7990) to (104.34, 103.54, 11.9) mm, rotated rx 180 ry 0 rz -180 deg; joints [0, 0, 0, 0, 0, 0]
  MoveL (T7991) to (104.34, 103.54, 10.1) mm, rotated rx 180 ry 0 rz -180 deg; joints [0, 0, 0, 0, 0, 0]
  Set speed (40.0 mm/s)
  Call Extruder 2.0
  MoveL (T7992) to (104.34, 103.54, 10.1) mm, rotated rx 180 ry 0 rz -180 deg; joints [0, 0, 0, 0, 0, 0]
  Set speed (26.5 mm/s)
  MoveL (T7993) to (104.34, 103.54, 10.1) mm, rotated rx 180 ry 0 rz -180 deg; joints [0, 0, 0, 0, 0, 0]
  Call Extruder 0.17274
  MoveL (T7994) to (110.01, 103.54, 10.1) mm, rotated rx 180 ry 0 rz -180 deg; joints [0, 0, 0, 0, 0, 0]
  Call Extruder 0.05778
  MoveL (T7995) to (110.01, 105.44, 10.1) mm, rotated rx 180 ry 0 rz -180 deg; joints [0, 0, 0, 0, 0, 0]
  Call Extruder 0.11724
  MoveL (T7996) to (113.86, 105.44, 10.1) mm, rotated rx 180 ry 0 rz -180 deg; joints [0, 0, 0, 0, 0, 0]
  Call Extruder 0.05778
  MoveL (T7997) to (113.86, 103.54, 10.1) mm, rotated rx 180 ry 0 rz -180 deg; joints [0, 0, 0, 0, 0, 0]
  Call Extruder 0.23155
  MoveL (T7998) to (121.46, 103.54, 10.1) mm, rotated rx 180 ry 0 rz -180 deg; joints [0, 0, 0, 0, 0, 0]
  Call Extruder 0.18952
  MoveL (T7999) to (121.46, 109.76, 10.1) mm, rotated rx 180 ry 0 rz -180 deg; joints [0, 0, 0, 0, 0, 0]
  Call Extruder 0.05895
  MoveL (T8000) to (119.53, 109.76, 10.1) mm, rotated rx 180 ry 0 rz -180 deg; joints [0, 0, 0, 0, 0, 0]
  Call Extruder 0.14201
  MoveL (T8001) to (119.52, 114.42, 10.1) mm, rotated rx 180 ry 0 rz -180 deg; joints [0, 0, 0, 0, 0, 0]
  Call Extruder 0.05901
  MoveL (T8002) to (121.46, 114.42, 10.1) mm, rotated rx 180 ry 0 rz -180 deg; joints [0, 0, 0, 0, 0, 0]
  Call Extruder 0.21434
  MoveL (T8003) to (121.46, 121.46, 10.1) mm, rotated rx 180 ry 0 rz -180 deg; joints [0, 0, 0, 0, 0, 0]
  Call Extruder 0.54596
  MoveL (T8004) to (103.54, 121.46, 10.1) mm, rotated rx 180 ry 0 rz -180 deg; joints [0, 0, 0, 0, 0, 0]
  Call Extruder 0.54596
  MoveL (T8005) to (103.54, 103.54, 10.1) mm, rotated rx 180 ry 0 rz -180 deg; joints [0, 0, 0, 0, 0, 0]
  Call Extruder 0.02254
  MoveL (T8006) to (104.28, 103.54, 10.1) mm, rotated rx 180 ry 0 rz -180 deg; joints [0, 0, 0, 0, 0, 0]
  Set speed (150.0 mm/s)
  MoveL (T8007) to (103.53, 103.13, 10.1) mm, rotated rx 180 ry 0 rz -180 deg; joints [0, 0, 0, 0, 0, 0]
  Set speed (26.5 mm/s)
  MoveL (T8008) to (103.53, 103.13, 10.1) mm, rotated rx 180 ry 0 rz -180 deg; joints [0, 0, 0, 0, 0, 0]
  Call Extruder 0.20972
  MoveL (T8009) to (110.42, 103.13, 10.1) mm, rotated rx 180 ry 0 rz -180 deg; joints [0, 0, 0, 0, 0, 0]
  Call Extruder 0.05778
  MoveL (T8010) to (110.42, 105.03, 10.1) mm, rotated rx 180 ry 0 rz -180 deg; joints [0, 0, 0, 0, 0, 0]
  Call Extruder 0.09245
  MoveL (T8011) to (113.45, 105.03, 10.1) mm, rotated rx 180 ry 0 rz -180 deg; joints [0, 0, 0, 0, 0, 0]
  Call Extruder 0.05778
  MoveL (T8012) to (113.45, 103.13, 10.1) mm, rotated rx 180 ry 0 rz -180 deg; joints [0, 0, 0, 0, 0, 0]
  Call Extruder 0.25635
  MoveL (T8013) to (121.87, 103.13, 10.1) mm, rotated rx 180 ry 0 rz -180 deg; joints [0, 0, 0, 0, 0, 0]
  Call Extruder 0.21431
  MoveL (T8014) to (121.87, 110.17, 10.1) mm, rotated rx 180 ry 0 rz -180 deg; joints [0, 0, 0, 0, 0, 0]
  Call Extruder 0.05896
  MoveL (T8015) to (119.93, 110.17, 10.1) mm, rotated rx 180 ry 0 rz -180 deg; joints [0, 0, 0, 0, 0, 0]
  Call Extruder 0.11723
  MoveL (T8016) to (119.93, 114.02, 10.1) mm, rotated rx 180 ry 0 rz -180 deg; joints [0, 0, 0, 0, 0, 0]
  Call Extruder 0.05901
  MoveL (T8017) to (121.87, 114.02, 10.1) mm, rotated rx 180 ry 0 rz -180 deg; joints [0, 0, 0, 0, 0, 0]
  Call Extruder 0.23912
  MoveL (T8018) to (121.87, 121.87, 10.1) mm, rotated rx 180 ry 0 rz -180 deg; joints [0, 0, 0, 0, 0, 0]
  Call Extruder 0.57077
  MoveL (T8019) to (103.13, 121.87, 10.1) mm, rotated rx 180 ry 0 rz -180 deg; joints [0, 0, 0, 0, 0, 0]
  Call Extruder 0.57077
  MoveL (T8020) to (103.13, 103.13, 10.1) mm, rotated rx 180 ry 0 rz -180 deg; joints [0, 0, 0, 0, 0, 0]
  Call Extruder 0.01036
  MoveL (T8021) to (103.47, 103.13, 10.1) mm, rotated rx 180 ry 0 rz -180 deg; joints [0, 0, 0, 0, 0, 0]
  Set speed (150.0 mm/s)
  MoveL (T8022) to (102.72, 102.81, 10.1) mm, rotated rx 180 ry 0 rz -180 deg; joints [0, 0, 0, 0, 0, 0]
  Set speed (25.0 mm/s)
  MoveL (T8023) to (102.72, 102.81, 10.1) mm, rotated rx 180 ry 0 rz -180 deg; joints [0, 0, 0, 0, 0, 0]
  Call Extruder 0.00259
  MoveL (T8024) to (102.72, 102.72, 10.1) mm, rotated rx 180 ry 0 rz -180 deg; joints [0, 0, 0, 0, 0, 0]
  Call Extruder 0.2467
  MoveL (T8025) to (110.82, 102.72, 10.1) mm, rotated rx 180 ry 0 rz -180 deg; joints [0, 0, 0, 0, 0, 0]
  Call Extruder 0.05778
  MoveL (T8026) to (110.82, 104.62, 10.1) mm, rotated rx 180 ry 0 rz -180 deg; joints [0, 0, 0, 0, 0, 0]
  Call Extruder 0.06766
  MoveL (T8027) to (113.05, 104.62, 10.1) mm, rotated rx 180 ry 0 rz -180 deg; joints [0, 0, 0, 0, 0, 0]
  Call Extruder 0.05778
  MoveL (T8028) to (113.05, 102.72, 10.1) mm, rotated rx 180 ry 0 rz -180 deg; joints [0, 0, 0, 0, 0, 0]
  Call Extruder 0.28115
  MoveL (T8029) to (122.28, 102.72, 10.1) mm, rotated rx 180 ry 0 rz -180 deg; joints [0, 0, 0, 0, 0, 0]
  Call Extruder 0.23911
  MoveL (T8030) to (122.28, 110.57, 10.1) mm, rotated rx 180 ry 0 rz -180 deg; joints [0, 0, 0, 0, 0, 0]
  Call Extruder 0.05896
  MoveL (T8031) to (120.34, 110.58, 10.1) mm, rotated rx 180 ry 0 rz -180 deg; joints [0, 0, 0, 0, 0, 0]
  Call Extruder 0.09244
  MoveL (T8032) to (120.34, 113.61, 10.1) mm, rotated rx 180 ry 0 rz -180 deg; joints [0, 0, 0, 0, 0, 0]
  Call Extruder 0.059
  MoveL (T8033) to (122.28, 113.61, 10.1) mm, rotated rx 180 ry 0 rz -180 deg; joints [0, 0, 0, 0, 0, 0]
  Call Extruder 0.26391
  MoveL (T8034) to (122.28, 122.28, 10.1) mm, rotated rx 180 ry 0 rz -180 deg; joints [0, 0, 0, 0, 0, 0]
  Call Extruder 0.59557
  MoveL (T8035) to (102.72, 122.28, 10.1) mm, rotated rx 180 ry 0 rz -180 deg; joints [0, 0, 0, 0, 0, 0]
  Call Extruder 0.59115
  MoveL (T8036) to (102.72, 102.87, 10.1) mm, rotated rx 180 ry 0 rz -180 deg; joints [0, 0, 0, 0, 0, 0]
  Set speed (150.0 mm/s)
  MoveL (T8037) to (102.78, 102.75, 10.1) mm, rotated rx 180 ry 0 rz -180 deg; joints [0, 0, 0, 0, 0, 0]
  Set speed (45.0 mm/s)
  Call Extruder -1.6
  MoveL (T8038) to (102.78, 102.75, 10.1) mm, rotated rx 180 ry 0 rz -180 deg; joints [0, 0, 0, 0, 0, 0]
  Set speed (120.0 mm/s)
  MoveL (T8039) to (102.78, 102.75, 10.1) mm, rotated rx 180 ry 0 rz -180 deg; joints [0, 0, 0, 0, 0, 0]
  Call Extruder -0.05166
  MoveL (T8040) to (102.72, 102.72, 10.1) mm, rotated rx 180 ry 0 rz -180 deg; joints [0, 0, 0, 0, 0, 0]
  Call Extruder -0.32834
  MoveL (T8041) to (103.65, 102.72, 10.1) mm, rotated rx 180 ry 0 rz -180 deg; joints [0, 0, 0, 0, 0, 0]
  Set speed (45.0 mm/s)
  Call Extruder -0.02
  MoveL (T8042) to (103.65, 102.72, 10.1) mm, rotated rx 180 ry 0 rz -180 deg; joints [0, 0, 0, 0, 0, 0]
  Set speed (150.0 mm/s)
  MoveL (T8043) to (103.65, 102.72, 12.1) mm, rotated rx 180 ry 0 rz -180 deg; joints [0, 0, 0, 0, 0, 0]
  MoveL (T8044) to (106.29, 103.84, 12.1) mm, rotated rx 180 ry 0 rz -180 deg; joints [0, 0, 0, 0, 0, 0]
  MoveL (T8045) to (106.29, 103.84, 10.1) mm, rotated rx 180 ry 0 rz -180 deg; joints [0, 0, 0, 0, 0, 0]
  Set speed (40.0 mm/s)
  Call Extruder 2.0
  MoveL (T8046) to (106.29, 103.84, 10.1) mm, rotated rx 180 ry 0 rz -180 deg; joints [0, 0, 0, 0, 0, 0]
  Set speed (26.5 mm/s)
  MoveL (T8047) to (106.29, 103.84, 10.1) mm, rotated rx 180 ry 0 rz -180 deg; joints [0, 0, 0, 0, 0, 0]
  Call Extruder 0.07441
  MoveL (T8048) to (103.84, 103.84, 10.1) mm, rotated rx 180 ry 0 rz -180 deg; joints [0, 0, 0, 0, 0, 0]
  Call Extruder 0.7458
  MoveL (T8049) to (121.16, 121.16, 10.1) mm, rotated rx 180 ry 0 rz -180 deg; joints [0, 0, 0, 0, 0, 0]
  Call Extruder 0.07441
  MoveL (T8050) to (118.71, 121.16, 10.1) mm, rotated rx 180 ry 0 rz -180 deg; joints [0, 0, 0, 0, 0, 0]
  Set speed (45.0 mm/s)
  Call Extruder -1.6
  MoveL (T8051) to (118.71, 121.16, 10.1) mm, rotated rx 180 ry 0 rz -180 deg; joints [0, 0, 0, 0, 0, 0]
  Set speed (120.0 mm/s)
  MoveL (T8052) to (118.71, 121.16, 10.1) mm, rotated rx 180 ry 0 rz -180 deg; joints [0, 0, 0, 0, 0, 0]
  Call Extruder -0.38
  MoveL (T8053) to (119.78, 121.16, 10.1) mm, rotated rx 180 ry 0 rz -180 deg; joints [0, 0, 0, 0, 0, 0]
  Set speed (45.0 mm/s)
  Call Extruder -0.02
  MoveL (T8054) to (119.78, 121.16, 10.1) mm, rotated rx 180 ry 0 rz -180 deg; joints [0, 0, 0, 0, 0, 0]
  Set speed (150.0 mm/s)
  MoveL (T8055) to (119.78, 121.16, 12.1) mm, rotated rx 180 ry 0 rz -180 deg; joints [0, 0, 0, 0, 0, 0]
  MoveL (T8056) to (121.16, 116.35, 12.1) mm, rotated rx 180 ry 0 rz -180 deg; joints [0, 0, 0, 0, 0, 0]
  MoveL (T8057) to (121.16, 116.35, 10.1) mm, rotated rx 180 ry 0 rz -180 deg; joints [0, 0, 0, 0, 0, 0]
  Set speed (40.0 mm/s)
  Call Extruder 2.0
  MoveL (T8058) to (121.16, 116.35, 10.1) mm, rotated rx 180 ry 0 rz -180 deg; joints [0, 0, 0, 0, 0, 0]
  Set speed (26.5 mm/s)
  MoveL (T8059) to (121.16, 116.35, 10.1) mm, rotated rx 180 ry 0 rz -180 deg; joints [0, 0, 0, 0, 0, 0]
  Call Extruder 0.02462
  MoveL (T8060) to (121.16, 115.54, 10.1) mm, rotated rx 180 ry 0 rz -180 deg; joints [0, 0, 0, 0, 0, 0]
  Call Extruder 0.03087
  MoveL (T8061) to (120.14, 115.54, 10.1) mm, rotated rx 180 ry 0 rz -180 deg; joints [0, 0, 0, 0, 0, 0]
  Call Extruder 0.04365
  MoveL (T8062) to (121.16, 116.55, 10.1) mm, rotated rx 180 ry 0 rz -180 deg; joints [0, 0, 0, 0, 0, 0]
  Call Extruder 0.03385
  MoveL (T8063) to (121.16, 117.66, 10.1) mm, rotated rx 180 ry 0 rz -180 deg; joints [0, 0, 0, 0, 0, 0]
  Call Extruder 0.15054
  MoveL (T8064) to (117.66, 121.16, 10.1) mm, rotated rx 180 ry 0 rz -180 deg; joints [0, 0, 0, 0, 0, 0]
  Call Extruder 0.03385
  MoveL (T8065) to (116.55, 121.16, 10.1) mm, rotated rx 180 ry 0 rz -180 deg; joints [0, 0, 0, 0, 0, 0]
  Call Extruder 0.54738
  MoveL (T8066) to (103.84, 108.45, 10.1) mm, rotated rx 180 ry 0 rz -180 deg; joints [0, 0, 0, 0, 0, 0]
  Call Extruder 0.03385
  MoveL (T8067) to (103.84, 107.34, 10.1) mm, rotated rx 180 ry 0 rz -180 deg; joints [0, 0, 0, 0, 0, 0]
  Call Extruder 0.15054
  MoveL (T8068) to (107.34, 103.84, 10.1) mm, rotated rx 180 ry 0 rz -180 deg; joints [0, 0, 0, 0, 0, 0]
  Call Extruder 0.03385
  MoveL (T8069) to (108.45, 103.84, 10.1) mm, rotated rx 180 ry 0 rz -180 deg; joints [0, 0, 0, 0, 0, 0]
  Call Extruder 0.02262
  MoveL (T8070) to (108.97, 104.37, 10.1) mm, rotated rx 180 ry 0 rz -180 deg; joints [0, 0, 0, 0, 0, 0]
  Call Extruder 0.03598
  MoveL (T8071) to (108.97, 105.55, 10.1) mm, rotated rx 180 ry 0 rz -180 deg; joints [0, 0, 0, 0, 0, 0]
  Call Extruder 0.01377
  MoveL (T8072) to (109.29, 105.87, 10.1) mm, rotated rx 180 ry 0 rz -180 deg; joints [0, 0, 0, 0, 0, 0]
  Call Extruder 0.01282
  MoveL (T8073) to (109.72, 105.87, 10.1) mm, rotated rx 180 ry 0 rz -180 deg; joints [0, 0, 0, 0, 0, 0]
  Set speed (150.0 mm/s)
  MoveL (T8074) to (109.2, 105.33, 10.1) mm, rotated rx 180 ry 0 rz -180 deg; joints [0, 0, 0, 0, 0, 0]
  Set speed (26.5 mm/s)
  MoveL (T8075) to (109.2, 105.33, 10.1) mm, rotated rx 180 ry 0 rz -180 deg; joints [0, 0, 0, 0, 0, 0]
  Call Extruder 0.02473
  MoveL (T8076) to (109.7, 104.82, 10.1) mm, rotated rx 180 ry 0 rz -180 deg; joints [0, 0, 0, 0, 0, 0]
  Call Extruder 0.02254
  MoveL (T8077) to (109.7, 104.17, 10.1) mm, rotated rx 180 ry 0 rz -180 deg; joints [0, 0, 0, 0, 0, 0]
  Call Extruder 0.0247
  MoveL (T8078) to (109.2, 104.67, 10.1) mm, rotated rx 180 ry 0 rz -180 deg; joints [0, 0, 0, 0, 0, 0]
  Set speed (45.0 mm/s)
  Call Extruder -1.6
  MoveL (T8079) to (109.2, 104.67, 10.1) mm, rotated rx 180 ry 0 rz -180 deg; joints [0, 0, 0, 0, 0, 0]
  Set speed (120.0 mm/s)
  MoveL (T8080) to (109.2, 104.67, 10.1) mm, rotated rx 180 ry 0 rz -180 deg; joints [0, 0, 0, 0, 0, 0]
  Call Extruder -0.25469
  MoveL (T8081) to (109.7, 104.17, 10.1) mm, rotated rx 180 ry 0 rz -180 deg; joints [0, 0, 0, 0, 0, 0]
  Call Extruder -0.12531
  MoveL (T8082) to (109.7, 104.52, 10.1) mm, rotated rx 180 ry 0 rz -180 deg; joints [0, 0, 0, 0, 0, 0]
  Set speed (45.0 mm/s)
  Call Extruder -0.02
  MoveL (T8083) to (109.7, 104.52, 10.1) mm, rotated rx 180 ry 0 rz -180 deg; joints [0, 0, 0, 0, 0, 0]
  Set speed (150.0 mm/s)
  MoveL (T8084) to (109.7, 104.52, 12.1) mm, rotated rx 180 ry 0 rz -180 deg; joints [0, 0, 0, 0, 0, 0]
  MoveL (T8085) to (112.14, 105.74, 12.1) mm, rotated rx 180 ry 0 rz -180 deg; joints [0, 0, 0, 0, 0, 0]
  MoveL (T8086) to (112.14, 105.74, 10.1) mm, rotated rx 180 ry 0 rz -180 deg; joints [0, 0, 0, 0, 0, 0]
  Set speed (40.0 mm/s)
  Call Extruder 2.0
  MoveL (T8087) to (112.14, 105.74, 10.1) mm, rotated rx 180 ry 0 rz -180 deg; joints [0, 0, 0, 0, 0, 0]
  Set speed (26.5 mm/s)
  MoveL (T8088) to (112.14, 105.74, 10.1) mm, rotated rx 180 ry 0 rz -180 deg; joints [0, 0, 0, 0, 0, 0]
  Call Extruder 0.0513
  MoveL (T8089) to (113.82, 105.74, 10.1) mm, rotated rx 180 ry 0 rz -180 deg; joints [0, 0, 0, 0, 0, 0]
  Call Extruder 0.00557
  MoveL (T8090) to (113.95, 105.87, 10.1) mm, rotated rx 180 ry 0 rz -180 deg; joints [0, 0, 0, 0, 0, 0]
  Call Extruder 0.01754
  MoveL (T8091) to (114.52, 105.87, 10.1) mm, rotated rx 180 ry 0 rz -180 deg; joints [0, 0, 0, 0, 0, 0]
  Call Extruder 0.46011
  MoveL (T8092) to (103.84, 116.55, 10.1) mm, rotated rx 180 ry 0 rz -180 deg; joints [0, 0, 0, 0, 0, 0]
  Call Extruder 0.03385
  MoveL (T8093) to (103.84, 117.66, 10.1) mm, rotated rx 180 ry 0 rz -180 deg; joints [0, 0, 0, 0, 0, 0]
  Call Extruder 0.15054
  MoveL (T8094) to (107.34, 121.16, 10.1) mm, rotated rx 180 ry 0 rz -180 deg; joints [0, 0, 0, 0, 0, 0]
  Call Extruder 0.03385
  MoveL (T8095) to (108.45, 121.16, 10.1) mm, rotated rx 180 ry 0 rz -180 deg; joints [0, 0, 0, 0, 0, 0]
  Call Extruder 0.464
  MoveL (T8096) to (119.22, 110.39, 10.1) mm, rotated rx 180 ry 0 rz -180 deg; joints [0, 0, 0, 0, 0, 0]
  Call Extruder 0.01146
  MoveL (T8097) to (119.22, 110.01, 10.1) mm, rotated rx 180 ry 0 rz -180 deg; joints [0, 0, 0, 0, 0, 0]
  Call Extruder 0.1862
  MoveL (T8098) to (114.9, 105.69, 10.1) mm, rotated rx 180 ry 0 rz -180 deg; joints [0, 0, 0, 0, 0, 0]
  Call Extruder 0.00588
  MoveL (T8099) to (115.03, 105.55, 10.1) mm, rotated rx 180 ry 0 rz -180 deg; joints [0, 0, 0, 0, 0, 0]
  Call Extruder 0.00582
  MoveL (T8100) to (115.03, 105.36, 10.1) mm, rotated rx 180 ry 0 rz -180 deg; joints [0, 0, 0, 0, 0, 0]
  Call Extruder 0.06528
  MoveL (T8101) to (116.55, 103.84, 10.1) mm, rotated rx 180 ry 0 rz -180 deg; joints [0, 0, 0, 0, 0, 0]
  Call Extruder 0.03385
  MoveL (T8102) to (117.66, 103.84, 10.1) mm, rotated rx 180 ry 0 rz -180 deg; joints [0, 0, 0, 0, 0, 0]
  Call Extruder 0.15054
  MoveL (T8103) to (121.16, 107.34, 10.1) mm, rotated rx 180 ry 0 rz -180 deg; joints [0, 0, 0, 0, 0, 0]
  Call Extruder 0.03385
  MoveL (T8104) to (121.16, 108.45, 10.1) mm, rotated rx 180 ry 0 rz -180 deg; joints [0, 0, 0, 0, 0, 0]
  Call Extruder 0.00686
  MoveL (T8105) to (121, 108.61, 10.1) mm, rotated rx 180 ry 0 rz -180 deg; joints [0, 0, 0, 0, 0, 0]
  Call Extruder 0.04822
  MoveL (T8106) to (119.41, 108.61, 10.1) mm, rotated rx 180 ry 0 rz -180 deg; joints [0, 0, 0, 0, 0, 0]
  Call Extruder 0.01373
  MoveL (T8107) to (119.09, 108.93, 10.1) mm, rotated rx 180 ry 0 rz -180 deg; joints [0, 0, 0, 0, 0, 0]
  Call Extruder 0.01246
  MoveL (T8108) to (119.09, 109.34, 10.1) mm, rotated rx 180 ry 0 rz -180 deg; joints [0, 0, 0, 0, 0, 0]
  Set speed (45.0 mm/s)
  Call Extruder -1.6
  MoveL (T8109) to (119.09, 109.34, 10.1) mm, rotated rx 180 ry 0 rz -180 deg; joints [0, 0, 0, 0, 0, 0]
  Set speed (120.0 mm/s)
  MoveL (T8110) to (119.09, 109.34, 10.1) mm, rotated rx 180 ry 0 rz -180 deg; joints [0, 0, 0, 0, 0, 0]
  Call Extruder -0.14568
  MoveL (T8111) to (119.09, 108.93, 10.1) mm, rotated rx 180 ry 0 rz -180 deg; joints [0, 0, 0, 0, 0, 0]
  Call Extruder -0.16059
  MoveL (T8112) to (119.41, 108.61, 10.1) mm, rotated rx 180 ry 0 rz -180 deg; joints [0, 0, 0, 0, 0, 0]
  Call Extruder -0.07373
  MoveL (T8113) to (119.62, 108.61, 10.1) mm, rotated rx 180 ry 0 rz -180 deg; joints [0, 0, 0, 0, 0, 0]
  Set speed (45.0 mm/s)
  Call Extruder -0.02
  MoveL (T8114) to (119.62, 108.61, 10.1) mm, rotated rx 180 ry 0 rz -180 deg; joints [0, 0, 0, 0, 0, 0]
  Set speed (150.0 mm/s)
  MoveL (T8115) to (119.62, 108.61, 12.1) mm, rotated rx 180 ry 0 rz -180 deg; joints [0, 0, 0, 0, 0, 0]
  MoveL (T8116) to (121.17, 108.83, 12.1) mm, rotated rx 180 ry 0 rz -180 deg; joints [0, 0, 0, 0, 0, 0]
  MoveL (T8117) to (121.17, 108.83, 10.1) mm, rotated rx 180 ry 0 rz -180 deg; joints [0, 0, 0, 0, 0, 0]
  Set speed (40.0 mm/s)
  Call Extruder 2.0
  MoveL (T8118) to (121.17, 108.83, 10.1) mm, rotated rx 180 ry 0 rz -180 deg; joints [0, 0, 0, 0, 0, 0]
  Set speed (26.5 mm/s)
  MoveL (T8119) to (121.17, 108.83, 10.1) mm, rotated rx 180 ry 0 rz -180 deg; joints [0, 0, 0, 0, 0, 0]
  Call Extruder 0.03151
  MoveL (T8120) to (120.55, 109.45, 10.1) mm, rotated rx 180 ry 0 rz -180 deg; joints [0, 0, 0, 0, 0, 0]
  Call Extruder 0.02424
  MoveL (T8121) to (119.87, 109.46, 10.1) mm, rotated rx 180 ry 0 rz -180 deg; joints [0, 0, 0, 0, 0, 0]
  Call Extruder 0.02223
  MoveL (T8122) to (120.31, 109.02, 10.1) mm, rotated rx 180 ry 0 rz -180 deg; joints [0, 0, 0, 0, 0, 0]
  Call Extruder 0.02424
  MoveL (T8123) to (119.63, 109.02, 10.1) mm, rotated rx 180 ry 0 rz -180 deg; joints [0, 0, 0, 0, 0, 0]
  Call Extruder 0.01595
  MoveL (T8124) to (119.32, 109.33, 10.1) mm, rotated rx 180 ry 0 rz -180 deg; joints [0, 0, 0, 0, 0, 0]
  Set speed (45.0 mm/s)
  Call Extruder -1.6
  MoveL (T8125) to (119.32, 109.33, 10.1) mm, rotated rx 180 ry 0 rz -180 deg; joints [0, 0, 0, 0, 0, 0]
  Set speed (120.0 mm/s)
  MoveL (T8126) to (119.32, 109.33, 10.1) mm, rotated rx 180 ry 0 rz -180 deg; joints [0, 0, 0, 0, 0, 0]
  Call Extruder -0.15869
  MoveL (T8127) to (119.63, 109.02, 10.1) mm, rotated rx 180 ry 0 rz -180 deg; joints [0, 0, 0, 0, 0, 0]
  Call Extruder -0.22131
  MoveL (T8128) to (120.25, 109.02, 10.1) mm, rotated rx 180 ry 0 rz -180 deg; joints [0, 0, 0, 0, 0, 0]
  Set speed (45.0 mm/s)
  Call Extruder -0.02
  MoveL (T8129) to (120.25, 109.02, 10.1) mm, rotated rx 180 ry 0 rz -180 deg; joints [0, 0, 0, 0, 0, 0]
  Set speed (150.0 mm/s)
  MoveL (T8130) to (120.25, 109.02, 12.1) mm, rotated rx 180 ry 0 rz -180 deg; joints [0, 0, 0, 0, 0, 0]
  MoveL (T8131) to (118.71, 103.84, 12.1) mm, rotated rx 180 ry 0 rz -180 deg; joints [0, 0, 0, 0, 0, 0]
  MoveL (T8132) to (118.71, 103.84, 10.1) mm, rotated rx 180 ry 0 rz -180 deg; joints [0, 0, 0, 0, 0, 0]
  Set speed (40.0 mm/s)
  Call Extruder 2.0
  MoveL (T8133) to (118.71, 103.84, 10.1) mm, rotated rx 180 ry 0 rz -180 deg; joints [0, 0, 0, 0, 0, 0]
  Set speed (26.5 mm/s)
  MoveL (T8134) to (118.71, 103.84, 10.1) mm, rotated rx 180 ry 0 rz -180 deg; joints [0, 0, 0, 0, 0, 0]
  Call Extruder 0.07441
  MoveL (T8135) to (121.16, 103.84, 10.1) mm, rotated rx 180 ry 0 rz -180 deg; joints [0, 0, 0, 0, 0, 0]
  Call Extruder 0.7458
  MoveL (T8136) to (103.84, 121.16, 10.1) mm, rotated rx 180 ry 0 rz -180 deg; joints [0, 0, 0, 0, 0, 0]
  Call Extruder 0.07441
  MoveL (T8137) to (106.29, 121.16, 10.1) mm, rotated rx 180 ry 0 rz -180 deg; joints [0, 0, 0, 0, 0, 0]
  Set speed (45.0 mm/s)
  Call Extruder -1.6
  MoveL (T8138) to (106.29, 121.16, 10.1) mm, rotated rx 180 ry 0 rz -180 deg; joints [0, 0, 0, 0, 0, 0]
  Set speed (120.0 mm/s)
  MoveL (T8139) to (106.29, 121.16, 10.1) mm, rotated rx 180 ry 0 rz -180 deg; joints [0, 0, 0, 0, 0, 0]
  Call Extruder -0.38
  MoveL (T8140) to (105.22, 121.16, 10.1) mm, rotated rx 180 ry 0 rz -180 deg; joints [0, 0, 0, 0, 0, 0]
  Set speed (45.0 mm/s)
  Call Extruder -0.02
  MoveL (T8141) to (105.22, 121.16, 10.1) mm, rotated rx 180 ry 0 rz -180 deg; joints [0, 0, 0, 0, 0, 0]
  Set speed (150.0 mm/s)
  MoveL (T8142) to (105.22, 121.16, 12.1) mm, rotated rx 180 ry 0 rz -180 deg; joints [0, 0, 0, 0, 0, 0]
  MoveL (T8143) to (103.84, 115.5, 12.1) mm, rotated rx 180 ry 0 rz -180 deg; joints [0, 0, 0, 0, 0, 0]
  MoveL (T8144) to (103.84, 115.5, 10.1) mm, rotated rx 180 ry 0 rz -180 deg; joints [0, 0, 0, 0, 0, 0]
  Set speed (40.0 mm/s)
  Call Extruder 2.0
  MoveL (T8145) to (103.84, 115.5, 10.1) mm, rotated rx 180 ry 0 rz -180 deg; joints [0, 0, 0, 0, 0, 0]
  Set speed (26.5 mm/s)
  MoveL (T8146) to (103.84, 115.5, 10.1) mm, rotated rx 180 ry 0 rz -180 deg; joints [0, 0, 0, 0, 0, 0]
  Call Extruder 0.07441
  MoveL (T8147) to (103.84, 113.06, 10.1) mm, rotated rx 180 ry 0 rz -180 deg; joints [0, 0, 0, 0, 0, 0]
  Call Extruder 0.34896
  MoveL (T8148) to (111.94, 121.16, 10.1) mm, rotated rx 180 ry 0 rz -180 deg; joints [0, 0, 0, 0, 0, 0]
  Call Extruder 0.03385
  MoveL (T8149) to (113.06, 121.16, 10.1) mm, rotated rx 180 ry 0 rz -180 deg; joints [0, 0, 0, 0, 0, 0]
  Call Extruder 0.26005
  MoveL (T8150) to (119.09, 115.12, 10.1) mm, rotated rx 180 ry 0 rz -180 deg; joints [0, 0, 0, 0, 0, 0]
  Call Extruder 0.01848
  MoveL (T8151) to (119.09, 114.51, 10.1) mm, rotated rx 180 ry 0 rz -180 deg; joints [0, 0, 0, 0, 0, 0]
  Call Extruder 0.00061
  MoveL (T8152) to (119.1, 114.5, 10.1) mm, rotated rx 180 ry 0 rz -180 deg; joints [0, 0, 0, 0, 0, 0]
  Call Extruder 0.37731
  MoveL (T8153) to (110.35, 105.74, 10.1) mm, rotated rx 180 ry 0 rz -180 deg; joints [0, 0, 0, 0, 0, 0]
  Call Extruder 0.00904
  MoveL (T8154) to (110.05, 105.74, 10.1) mm, rotated rx 180 ry 0 rz -180 deg; joints [0, 0, 0, 0, 0, 0]
  Call Extruder 0.2673
  MoveL (T8155) to (103.84, 111.94, 10.1) mm, rotated rx 180 ry 0 rz -180 deg; joints [0, 0, 0, 0, 0, 0]
  Call Extruder 0.07441
  MoveL (T8156) to (103.84, 109.5, 10.1) mm, rotated rx 180 ry 0 rz -180 deg; joints [0, 0, 0, 0, 0, 0]
  Set speed (45.0 mm/s)
  Call Extruder -1.6
  MoveL (T8157) to (103.84, 109.5, 10.1) mm, rotated rx 180 ry 0 rz -180 deg; joints [0, 0, 0, 0, 0, 0]
  Set speed (120.0 mm/s)
  MoveL (T8158) to (103.84, 109.5, 10.1) mm, rotated rx 180 ry 0 rz -180 deg; joints [0, 0, 0, 0, 0, 0]
  Call Extruder -0.38
  MoveL (T8159) to (103.84, 110.57, 10.1) mm, rotated rx 180 ry 0 rz -180 deg; joints [0, 0, 0, 0, 0, 0]
  Set speed (45.0 mm/s)
  Call Extruder -0.02
  MoveL (T8160) to (103.84, 110.57, 10.1) mm, rotated rx 180 ry 0 rz -180 deg; joints [0, 0, 0, 0, 0, 0]
  Set speed (150.0 mm/s)
  MoveL (T8161) to (103.84, 110.57, 12.1) mm, rotated rx 180 ry 0 rz -180 deg; joints [0, 0, 0, 0, 0, 0]
  MoveL (T8162) to (114.81, 105.15, 12.1) mm, rotated rx 180 ry 0 rz -180 deg; joints [0, 0, 0, 0, 0, 0]
  MoveL (T8163) to (114.81, 105.15, 10.1) mm, rotated rx 180 ry 0 rz -180 deg; joints [0, 0, 0, 0, 0, 0]
  Set speed (40.0 mm/s)
  Call Extruder 2.0
  MoveL (T8164) to (114.81, 105.15, 10.1) mm, rotated rx 180 ry 0 rz -180 deg; joints [0, 0, 0, 0, 0, 0]
  Set speed (26.5 mm/s)
  MoveL (T8165) to (114.81, 105.15, 10.1) mm, rotated rx 180 ry 0 rz -180 deg; joints [0, 0, 0, 0, 0, 0]
  Call Extruder 0.01579
  MoveL (T8166) to (114.5, 105.46, 10.1) mm, rotated rx 180 ry 0 rz -180 deg; joints [0, 0, 0, 0, 0, 0]
  Call Extruder 0.01188
  MoveL (T8167) to (114.16, 105.46, 10.1) mm, rotated rx 180 ry 0 rz -180 deg; joints [0, 0, 0, 0, 0, 0]
  Call Extruder 0.01215
  MoveL (T8168) to (114.16, 105.12, 10.1) mm, rotated rx 180 ry 0 rz -180 deg; joints [0, 0, 0, 0, 0, 0]
  Call Extruder 0.02334
  MoveL (T8169) to (114.63, 104.66, 10.1) mm, rotated rx 180 ry 0 rz -180 deg; joints [0, 0, 0, 0, 0, 0]
  Call Extruder 0.02401
  MoveL (T8170) to (114.63, 103.99, 10.1) mm, rotated rx 180 ry 0 rz -180 deg; joints [0, 0, 0, 0, 0, 0]
  Call Extruder 0.03255
  MoveL (T8171) to (113.98, 104.63, 10.1) mm, rotated rx 180 ry 0 rz -180 deg; joints [0, 0, 0, 0, 0, 0]
  Set speed (45.0 mm/s)
  Call Extruder -1.6
  MoveL (T8172) to (113.98, 104.63, 10.1) mm, rotated rx 180 ry 0 rz -180 deg; joints [0, 0, 0, 0, 0, 0]
  Set speed (120.0 mm/s)
  MoveL (T8173) to (113.98, 104.63, 10.1) mm, rotated rx 180 ry 0 rz -180 deg; joints [0, 0, 0, 0, 0, 0]
  Call Extruder -0.32519
  MoveL (T8174) to (114.63, 103.99, 10.1) mm, rotated rx 180 ry 0 rz -180 deg; joints [0, 0, 0, 0, 0, 0]
  Call Extruder -0.05481
  MoveL (T8175) to (114.63, 104.14, 10.1) mm, rotated rx 180 ry 0 rz -180 deg; joints [0, 0, 0, 0, 0, 0]
  Set speed (45.0 mm/s)
  Call Extruder -0.02
  MoveL (T8176) to (114.63, 104.14, 10.1) mm, rotated rx 180 ry 0 rz -180 deg; joints [0, 0, 0, 0, 0, 0]
  Set speed (150.0 mm/s)
  MoveL (T8177) to (114.63, 104.14, 12.1) mm, rotated rx 180 ry 0 rz -180 deg; joints [0, 0, 0, 0, 0, 0]
  MoveL (T8178) to (121.34, 114.94, 12.1) mm, rotated rx 180 ry 0 rz -180 deg; joints [0, 0, 0, 0, 0, 0]
  MoveL (T8179) to (121.34, 114.94, 10.1) mm, rotated rx 180 ry 0 rz -180 deg; joints [0, 0, 0, 0, 0, 0]
  Set speed (40.0 mm/s)
  Call Extruder 2.0
  MoveL (T8180) to (121.34, 114.94, 10.1) mm, rotated rx 180 ry 0 rz -180 deg; joints [0, 0, 0, 0, 0, 0]
  Set speed (26.5 mm/s)
  MoveL (T8181) to (121.34, 114.94, 10.1) mm, rotated rx 180 ry 0 rz -180 deg; joints [0, 0, 0, 0, 0, 0]
  Call Extruder 0.00969
  MoveL (T8182) to (121.15, 115.13, 10.1) mm, rotated rx 180 ry 0 rz -180 deg; joints [0, 0, 0, 0, 0, 0]
  Call Extruder 0.02463
  MoveL (T8183) to (120.47, 115.13, 10.1) mm, rotated rx 180 ry 0 rz -180 deg; joints [0, 0, 0, 0, 0, 0]
  Call Extruder 0.02046
  MoveL (T8184) to (120.87, 114.73, 10.1) mm, rotated rx 180 ry 0 rz -180 deg; joints [0, 0, 0, 0, 0, 0]
  Call Extruder 0.02463
  MoveL (T8185) to (120.19, 114.73, 10.1) mm, rotated rx 180 ry 0 rz -180 deg; joints [0, 0, 0, 0, 0, 0]
  Call Extruder 0.02046
  MoveL (T8186) to (119.79, 115.13, 10.1) mm, rotated rx 180 ry 0 rz -180 deg; joints [0, 0, 0, 0, 0, 0]
  Call Extruder 0.00744
  MoveL (T8187) to (119.58, 115.13, 10.1) mm, rotated rx 180 ry 0 rz -180 deg; joints [0, 0, 0, 0, 0, 0]
  Call Extruder 0.00413
  MoveL (T8188) to (119.5, 115.05, 10.1) mm, rotated rx 180 ry 0 rz -180 deg; joints [0, 0, 0, 0, 0, 0]
  Call Extruder 0.01134
  MoveL (T8189) to (119.5, 114.73, 10.1) mm, rotated rx 180 ry 0 rz -180 deg; joints [0, 0, 0, 0, 0, 0]
  Call Extruder 0.00967
  MoveL (T8190) to (119.69, 114.55, 10.1) mm, rotated rx 180 ry 0 rz -180 deg; joints [0, 0, 0, 0, 0, 0]
  Set speed (45.0 mm/s)
  Call Extruder -1.6
  MoveL (T8191) to (119.69, 114.55, 10.1) mm, rotated rx 180 ry 0 rz -180 deg; joints [0, 0, 0, 0, 0, 0]
  Set speed (120.0 mm/s)
  MoveL (T8192) to (119.69, 114.55, 10.1) mm, rotated rx 180 ry 0 rz -180 deg; joints [0, 0, 0, 0, 0, 0]
  Call Extruder -0.0954
  MoveL (T8193) to (119.5, 114.73, 10.1) mm, rotated rx 180 ry 0 rz -180 deg; joints [0, 0, 0, 0, 0, 0]
  Call Extruder -0.11183
  MoveL (T8194) to (119.5, 115.05, 10.1) mm, rotated rx 180 ry 0 rz -180 deg; joints [0, 0, 0, 0, 0, 0]
  Call Extruder -0.04075
  MoveL (T8195) to (119.58, 115.13, 10.1) mm, rotated rx 180 ry 0 rz -180 deg; joints [0, 0, 0, 0, 0, 0]
  Call Extruder -0.07339
  MoveL (T8196) to (119.79, 115.13, 10.1) mm, rotated rx 180 ry 0 rz -180 deg; joints [0, 0, 0, 0, 0, 0]
  Call Extruder -0.05863
  MoveL (T8197) to (119.9, 115.01, 10.1) mm, rotated rx 180 ry 0 rz -180 deg; joints [0, 0, 0, 0, 0, 0]
  Set speed (45.0 mm/s)
  Call Extruder -0.02
  MoveL (T8198) to (119.9, 115.01, 10.1) mm, rotated rx 180 ry 0 rz -180 deg; joints [0, 0, 0, 0, 0, 0]
  Set speed (150.0 mm/s)
  MoveL (T8199) to (119.9, 115.01, 12.1) mm, rotated rx 180 ry 0 rz -180 deg; joints [0, 0, 0, 0, 0, 0]
  MoveL (T8200) to (104.34, 103.54, 12.1) mm, rotated rx 180 ry 0 rz -180 deg; joints [0, 0, 0, 0, 0, 0]
  MoveL (T8201) to (104.34, 103.54, 10.3) mm, rotated rx 180 ry 0 rz -180 deg; joints [0, 0, 0, 0, 0, 0]
  Set speed (40.0 mm/s)
  Call Extruder 2.0
  MoveL (T8202) to (104.34, 103.54, 10.3) mm, rotated rx 180 ry 0 rz -180 deg; joints [0, 0, 0, 0, 0, 0]
  Set speed (26.7 mm/s)
  MoveL (T8203) to (104.34, 103.54, 10.3) mm, rotated rx 180 ry 0 rz -180 deg; joints [0, 0, 0, 0, 0, 0]
  Call Extruder 0.17158
  MoveL (T8204) to (109.97, 103.54, 10.3) mm, rotated rx 180 ry 0 rz -180 deg; joints [0, 0, 0, 0, 0, 0]
  Call Extruder 0.05778
  MoveL (T8205) to (109.97, 105.44, 10.3) mm, rotated rx 180 ry 0 rz -180 deg; joints [0, 0, 0, 0, 0, 0]
  Call Extruder 0.1216
  MoveL (T8206) to (113.96, 105.44, 10.3) mm, rotated rx 180 ry 0 rz -180 deg; joints [0, 0, 0, 0, 0, 0]
  Call Extruder 0.05778
  MoveL (T8207) to (113.96, 103.54, 10.3) mm, rotated rx 180 ry 0 rz -180 deg; joints [0, 0, 0, 0, 0, 0]
  Call Extruder 0.22847
  MoveL (T8208) to (121.46, 103.54, 10.3) mm, rotated rx 180 ry 0 rz -180 deg; joints [0, 0, 0, 0, 0, 0]
  Call Extruder 0.18587
  MoveL (T8209) to (121.46, 109.64, 10.3) mm, rotated rx 180 ry 0 rz -180 deg; joints [0, 0, 0, 0, 0, 0]
  Call Extruder 0.05894
  MoveL (T8210) to (119.53, 109.64, 10.3) mm, rotated rx 180 ry 0 rz -180 deg; joints [0, 0, 0, 0, 0, 0]
  Call Extruder 0.1491
  MoveL (T8211) to (119.52, 114.54, 10.3) mm, rotated rx 180 ry 0 rz -180 deg; joints [0, 0, 0, 0, 0, 0]
  Call Extruder 0.05901
  MoveL (T8212) to (121.46, 114.54, 10.3) mm, rotated rx 180 ry 0 rz -180 deg; joints [0, 0, 0, 0, 0, 0]
  Call Extruder 0.21088
  MoveL (T8213) to (121.46, 121.46, 10.3) mm, rotated rx 180 ry 0 rz -180 deg; joints [0, 0, 0, 0, 0, 0]
  Call Extruder 0.54596
  MoveL (T8214) to (103.54, 121.46, 10.3) mm, rotated rx 180 ry 0 rz -180 deg; joints [0, 0, 0, 0, 0, 0]
  Call Extruder 0.54596
  MoveL (T8215) to (103.54, 103.54, 10.3) mm, rotated rx 180 ry 0 rz -180 deg; joints [0, 0, 0, 0, 0, 0]
  Call Extruder 0.02254
  MoveL (T8216) to (104.28, 103.54, 10.3) mm, rotated rx 180 ry 0 rz -180 deg; joints [0, 0, 0, 0, 0, 0]
  Set speed (150.0 mm/s)
  MoveL (T8217) to (103.53, 103.13, 10.3) mm, rotated rx 180 ry 0 rz -180 deg; joints [0, 0, 0, 0, 0, 0]
  Set speed (26.7 mm/s)
  MoveL (T8218) to (103.53, 103.13, 10.3) mm, rotated rx 180 ry 0 rz -180 deg; joints [0, 0, 0, 0, 0, 0]
  Call Extruder 0.20858
  MoveL (T8219) to (110.38, 103.13, 10.3) mm, rotated rx 180 ry 0 rz -180 deg; joints [0, 0, 0, 0, 0, 0]
  Call Extruder 0.05778
  MoveL (T8220) to (110.38, 105.03, 10.3) mm, rotated rx 180 ry 0 rz -180 deg; joints [0, 0, 0, 0, 0, 0]
  Call Extruder 0.09678
  MoveL (T8221) to (113.56, 105.03, 10.3) mm, rotated rx 180 ry 0 rz -180 deg; joints [0, 0, 0, 0, 0, 0]
  Call Extruder 0.05778
  MoveL (T8222) to (113.55, 103.13, 10.3) mm, rotated rx 180 ry 0 rz -180 deg; joints [0, 0, 0, 0, 0, 0]
  Call Extruder 0.25328
  MoveL (T8223) to (121.87, 103.13, 10.3) mm, rotated rx 180 ry 0 rz -180 deg; joints [0, 0, 0, 0, 0, 0]
  Call Extruder 0.21067
  MoveL (T8224) to (121.87, 110.05, 10.3) mm, rotated rx 180 ry 0 rz -180 deg; joints [0, 0, 0, 0, 0, 0]
  Call Extruder 0.05895
  MoveL (T8225) to (119.93, 110.05, 10.3) mm, rotated rx 180 ry 0 rz -180 deg; joints [0, 0, 0, 0, 0, 0]
  Call Extruder 0.12432
  MoveL (T8226) to (119.93, 114.13, 10.3) mm, rotated rx 180 ry 0 rz -180 deg; joints [0, 0, 0, 0, 0, 0]
  Call Extruder 0.059
  MoveL (T8227) to (121.87, 114.13, 10.3) mm, rotated rx 180 ry 0 rz -180 deg; joints [0, 0, 0, 0, 0, 0]
  Call Extruder 0.23567
  MoveL (T8228) to (121.87, 121.87, 10.3) mm, rotated rx 180 ry 0 rz -180 deg; joints [0, 0, 0, 0, 0, 0]
  Call Extruder 0.57077
  MoveL (T8229) to (103.13, 121.87, 10.3) mm, rotated rx 180 ry 0 rz -180 deg; joints [0, 0, 0, 0, 0, 0]
  Call Extruder 0.57077
  MoveL (T8230) to (103.13, 103.13, 10.3) mm, rotated rx 180 ry 0 rz -180 deg; joints [0, 0, 0, 0, 0, 0]
  Call Extruder 0.01036
  MoveL (T8231) to (103.47, 103.13, 10.3) mm, rotated rx 180 ry 0 rz -180 deg; joints [0, 0, 0, 0, 0, 0]
  Set speed (150.0 mm/s)
  MoveL (T8232) to (102.72, 102.81, 10.3) mm, rotated rx 180 ry 0 rz -180 deg; joints [0, 0, 0, 0, 0, 0]
  Set speed (25.0 mm/s)
  MoveL (T8233) to (102.72, 102.81, 10.3) mm, rotated rx 180 ry 0 rz -180 deg; joints [0, 0, 0, 0, 0, 0]
  Call Extruder 0.00259
  MoveL (T8234) to (102.72, 102.72, 10.3) mm, rotated rx 180 ry 0 rz -180 deg; joints [0, 0, 0, 0, 0, 0]
  Call Extruder 0.24557
  MoveL (T8235) to (110.79, 102.72, 10.3) mm, rotated rx 180 ry 0 rz -180 deg; joints [0, 0, 0, 0, 0, 0]
  Call Extruder 0.05778
  MoveL (T8236) to (110.78, 104.62, 10.3) mm, rotated rx 180 ry 0 rz -180 deg; joints [0, 0, 0, 0, 0, 0]
  Call Extruder 0.07197
  MoveL (T8237) to (113.15, 104.62, 10.3) mm, rotated rx 180 ry 0 rz -180 deg; joints [0, 0, 0, 0, 0, 0]
  Call Extruder 0.05778
  MoveL (T8238) to (113.15, 102.72, 10.3) mm, rotated rx 180 ry 0 rz -180 deg; joints [0, 0, 0, 0, 0, 0]
  Call Extruder 0.27809
  MoveL (T8239) to (122.28, 102.72, 10.3) mm, rotated rx 180 ry 0 rz -180 deg; joints [0, 0, 0, 0, 0, 0]
  Call Extruder 0.23547
  MoveL (T8240) to (122.28, 110.45, 10.3) mm, rotated rx 180 ry 0 rz -180 deg; joints [0, 0, 0, 0, 0, 0]
  Call Extruder 0.05895
  MoveL (T8241) to (120.34, 110.45, 10.3) mm, rotated rx 180 ry 0 rz -180 deg; joints [0, 0, 0, 0, 0, 0]
  Call Extruder 0.09954
  MoveL (T8242) to (120.34, 113.72, 10.3) mm, rotated rx 180 ry 0 rz -180 deg; joints [0, 0, 0, 0, 0, 0]
  Call Extruder 0.05899
  MoveL (T8243) to (122.28, 113.72, 10.3) mm, rotated rx 180 ry 0 rz -180 deg; joints [0, 0, 0, 0, 0, 0]
  Call Extruder 0.26046
  MoveL (T8244) to (122.28, 122.28, 10.3) mm, rotated rx 180 ry 0 rz -180 deg; joints [0, 0, 0, 0, 0, 0]
  Call Extruder 0.59557
  MoveL (T8245) to (102.72, 122.28, 10.3) mm, rotated rx 180 ry 0 rz -180 deg; joints [0, 0, 0, 0, 0, 0]
  Call Extruder 0.59115
  MoveL (T8246) to (102.72, 102.87, 10.3) mm, rotated rx 180 ry 0 rz -180 deg; joints [0, 0, 0, 0, 0, 0]
  Set speed (150.0 mm/s)
  MoveL (T8247) to (102.78, 102.75, 10.3) mm, rotated rx 180 ry 0 rz -180 deg; joints [0, 0, 0, 0, 0, 0]
  Set speed (45.0 mm/s)
  Call Extruder -1.6
  MoveL (T8248) to (102.78, 102.75, 10.3) mm, rotated rx 180 ry 0 rz -180 deg; joints [0, 0, 0, 0, 0, 0]
  Set speed (120.0 mm/s)
  MoveL (T8249) to (102.78, 102.75, 10.3) mm, rotated rx 180 ry 0 rz -180 deg; joints [0, 0, 0, 0, 0, 0]
  Call Extruder -0.05166
  MoveL (T8250) to (102.72, 102.72, 10.3) mm, rotated rx 180 ry 0 rz -180 deg; joints [0, 0, 0, 0, 0, 0]
  Call Extruder -0.32834
  MoveL (T8251) to (103.65, 102.72, 10.3) mm, rotated rx 180 ry 0 rz -180 deg; joints [0, 0, 0, 0, 0, 0]
  Set speed (45.0 mm/s)
  Call Extruder -0.02
  MoveL (T8252) to (103.65, 102.72, 10.3) mm, rotated rx 180 ry 0 rz -180 deg; joints [0, 0, 0, 0, 0, 0]
  Set speed (150.0 mm/s)
  MoveL (T8253) to (103.65, 102.72, 12.3) mm, rotated rx 180 ry 0 rz -180 deg; joints [0, 0, 0, 0, 0, 0]
  MoveL (T8254) to (106.29, 103.84, 12.3) mm, rotated rx 180 ry 0 rz -180 deg; joints [0, 0, 0, 0, 0, 0]
  MoveL (T8255) to (106.29, 103.84, 10.3) mm, rotated rx 180 ry 0 rz -180 deg; joints [0, 0, 0, 0, 0, 0]
  Set speed (40.0 mm/s)
  Call Extruder 2.0
  MoveL (T8256) to (106.29, 103.84, 10.3) mm, rotated rx 180 ry 0 rz -180 deg; joints [0, 0, 0, 0, 0, 0]
  Set speed (26.7 mm/s)
  MoveL (T8257) to (106.29, 103.84, 10.3) mm, rotated rx 180 ry 0 rz -180 deg; joints [0, 0, 0, 0, 0, 0]
  Call Extruder 0.07441
  MoveL (T8258) to (103.84, 103.84, 10.3) mm, rotated rx 180 ry 0 rz -180 deg; joints [0, 0, 0, 0, 0, 0]
  Call Extruder 0.7458
  MoveL (T8259) to (121.16, 121.16, 10.3) mm, rotated rx 180 ry 0 rz -180 deg; joints [0, 0, 0, 0, 0, 0]
  Call Extruder 0.07441
  MoveL (T8260) to (118.71, 121.16, 10.3) mm, rotated rx 180 ry 0 rz -180 deg; joints [0, 0, 0, 0, 0, 0]
  Set speed (45.0 mm/s)
  Call Extruder -1.6
  MoveL (T8261) to (118.71, 121.16, 10.3) mm, rotated rx 180 ry 0 rz -180 deg; joints [0, 0, 0, 0, 0, 0]
  Set speed (120.0 mm/s)
  MoveL (T8262) to (118.71, 121.16, 10.3) mm, rotated rx 180 ry 0 rz -180 deg; joints [0, 0, 0, 0, 0, 0]
  Call Extruder -0.38
  MoveL (T8263) to (119.78, 121.16, 10.3) mm, rotated rx 180 ry 0 rz -180 deg; joints [0, 0, 0, 0, 0, 0]
  Set speed (45.0 mm/s)
  Call Extruder -0.02
  MoveL (T8264) to (119.78, 121.16, 10.3) mm, rotated rx 180 ry 0 rz -180 deg; joints [0, 0, 0, 0, 0, 0]
  Set speed (150.0 mm/s)
  MoveL (T8265) to (119.78, 121.16, 12.3) mm, rotated rx 180 ry 0 rz -180 deg; joints [0, 0, 0, 0, 0, 0]
  MoveL (T8266) to (121.16, 116.35, 12.3) mm, rotated rx 180 ry 0 rz -180 deg; joints [0, 0, 0, 0, 0, 0]
  MoveL (T8267) to (121.16, 116.35, 10.3) mm, rotated rx 180 ry 0 rz -180 deg; joints [0, 0, 0, 0, 0, 0]
  Set speed (40.0 mm/s)
  Call Extruder 2.0
  MoveL (T8268) to (121.16, 116.35, 10.3) mm, rotated rx 180 ry 0 rz -180 deg; joints [0, 0, 0, 0, 0, 0]
  Set speed (26.7 mm/s)
  MoveL (T8269) to (121.16, 116.35, 10.3) mm, rotated rx 180 ry 0 rz -180 deg; joints [0, 0, 0, 0, 0, 0]
  Call Extruder 0.02117
  MoveL (T8270) to (121.16, 115.65, 10.3) mm, rotated rx 180 ry 0 rz -180 deg; joints [0, 0, 0, 0, 0, 0]
  Call Extruder 0.02741
  MoveL (T8271) to (120.26, 115.65, 10.3) mm, rotated rx 180 ry 0 rz -180 deg; joints [0, 0, 0, 0, 0, 0]
  Call Extruder 0.03876
  MoveL (T8272) to (121.16, 116.55, 10.3) mm, rotated rx 180 ry 0 rz -180 deg; joints [0, 0, 0, 0, 0, 0]
  Call Extruder 0.03385
  MoveL (T8273) to (121.16, 117.66, 10.3) mm, rotated rx 180 ry 0 rz -180 deg; joints [0, 0, 0, 0, 0, 0]
  Call Extruder 0.15054
  MoveL (T8274) to (117.66, 121.16, 10.3) mm, rotated rx 180 ry 0 rz -180 deg; joints [0, 0, 0, 0, 0, 0]
  Call Extruder 0.03385
  MoveL (T8275) to (116.55, 121.16, 10.3) mm, rotated rx 180 ry 0 rz -180 deg; joints [0, 0, 0, 0, 0, 0]
  Call Extruder 0.54738
  MoveL (T8276) to (103.84, 108.45, 10.3) mm, rotated rx 180 ry 0 rz -180 deg; joints [0, 0, 0, 0, 0, 0]
  Call Extruder 0.03385
  MoveL (T8277) to (103.84, 107.34, 10.3) mm, rotated rx 180 ry 0 rz -180 deg; joints [0, 0, 0, 0, 0, 0]
  Call Extruder 0.15054
  MoveL (T8278) to (107.34, 103.84, 10.3) mm, rotated rx 180 ry 0 rz -180 deg; joints [0, 0, 0, 0, 0, 0]
  Call Extruder 0.03385
  MoveL (T8279) to (108.45, 103.84, 10.3) mm, rotated rx 180 ry 0 rz -180 deg; joints [0, 0, 0, 0, 0, 0]
  Call Extruder 0.01778
  MoveL (T8280) to (108.86, 104.26, 10.3) mm, rotated rx 180 ry 0 rz -180 deg; joints [0, 0, 0, 0, 0, 0]
  Call Extruder 0.03941
  MoveL (T8281) to (108.86, 105.55, 10.3) mm, rotated rx 180 ry 0 rz -180 deg; joints [0, 0, 0, 0, 0, 0]
  Call Extruder 0.01377
  MoveL (T8282) to (109.18, 105.87, 10.3) mm, rotated rx 180 ry 0 rz -180 deg; joints [0, 0, 0, 0, 0, 0]
  Call Extruder 0.02123
  MoveL (T8283) to (109.88, 105.87, 10.3) mm, rotated rx 180 ry 0 rz -180 deg; joints [0, 0, 0, 0, 0, 0]
  Set speed (45.0 mm/s)
  Call Extruder -1.6
  MoveL (T8284) to (109.88, 105.87, 10.3) mm, rotated rx 180 ry 0 rz -180 deg; joints [0, 0, 0, 0, 0, 0]
  Set speed (120.0 mm/s)
  MoveL (T8285) to (109.88, 105.87, 10.3) mm, rotated rx 180 ry 0 rz -180 deg; joints [0, 0, 0, 0, 0, 0]
  Call Extruder -0.24825
  MoveL (T8286) to (109.18, 105.87, 10.3) mm, rotated rx 180 ry 0 rz -180 deg; joints [0, 0, 0, 0, 0, 0]
  Call Extruder -0.13175
  MoveL (T8287) to (108.92, 105.61, 10.3) mm, rotated rx 180 ry 0 rz -180 deg; joints [0, 0, 0, 0, 0, 0]
  Set speed (45.0 mm/s)
  Call Extruder -0.02
  MoveL (T8288) to (108.92, 105.61, 10.3) mm, rotated rx 180 ry 0 rz -180 deg; joints [0, 0, 0, 0, 0, 0]
  Set speed (150.0 mm/s)
  MoveL (T8289) to (108.92, 105.61, 12.3) mm, rotated rx 180 ry 0 rz -180 deg; joints [0, 0, 0, 0, 0, 0]
  MoveL (T8290) to (109.09, 103.84, 12.3) mm, rotated rx 180 ry 0 rz -180 deg; joints [0, 0, 0, 0, 0, 0]
  MoveL (T8291) to (109.09, 103.84, 10.3) mm, rotated rx 180 ry 0 rz -180 deg; joints [0, 0, 0, 0, 0, 0]
  Set speed (40.0 mm/s)
  Call Extruder 2.0
  MoveL (T8292) to (109.09, 103.84, 10.3) mm, rotated rx 180 ry 0 rz -180 deg; joints [0, 0, 0, 0, 0, 0]
  Set speed (26.7 mm/s)
  MoveL (T8293) to (109.09, 103.84, 10.3) mm, rotated rx 180 ry 0 rz -180 deg; joints [0, 0, 0, 0, 0, 0]
  Call Extruder 0.02848
  MoveL (T8294) to (109.67, 104.42, 10.3) mm, rotated rx 180 ry 0 rz -180 deg; joints [0, 0, 0, 0, 0, 0]
  Call Extruder 0.02286
  MoveL (T8295) to (109.67, 105.08, 10.3) mm, rotated rx 180 ry 0 rz -180 deg; joints [0, 0, 0, 0, 0, 0]
  Call Extruder 0.01947
  MoveL (T8296) to (109.27, 104.68, 10.3) mm, rotated rx 180 ry 0 rz -180 deg; joints [0, 0, 0, 0, 0, 0]
  Call Extruder 0.02286
  MoveL (T8297) to (109.27, 105.34, 10.3) mm, rotated rx 180 ry 0 rz -180 deg; joints [0, 0, 0, 0, 0, 0]
  Call Extruder 0.01501
  MoveL (T8298) to (109.57, 105.65, 10.3) mm, rotated rx 180 ry 0 rz -180 deg; joints [0, 0, 0, 0, 0, 0]
  Set speed (45.0 mm/s)
  Call Extruder -1.6
  MoveL (T8299) to (109.57, 105.65, 10.3) mm, rotated rx 180 ry 0 rz -180 deg; joints [0, 0, 0, 0, 0, 0]
  Set speed (120.0 mm/s)
  MoveL (T8300) to (109.57, 105.65, 10.3) mm, rotated rx 180 ry 0 rz -180 deg; joints [0, 0, 0, 0, 0, 0]
  Call Extruder -0.15367
  MoveL (T8301) to (109.27, 105.34, 10.3) mm, rotated rx 180 ry 0 rz -180 deg; joints [0, 0, 0, 0, 0, 0]
  Call Extruder -0.22633
  MoveL (T8302) to (109.27, 104.71, 10.3) mm, rotated rx 180 ry 0 rz -180 deg; joints [0, 0, 0, 0, 0, 0]
  Set speed (45.0 mm/s)
  Call Extruder -0.02
  MoveL (T8303) to (109.27, 104.71, 10.3) mm, rotated rx 180 ry 0 rz -180 deg; joints [0, 0, 0, 0, 0, 0]
  Set speed (150.0 mm/s)
  MoveL (T8304) to (109.27, 104.71, 12.3) mm, rotated rx 180 ry 0 rz -180 deg; joints [0, 0, 0, 0, 0, 0]
  MoveL (T8305) to (114.56, 103.66, 12.3) mm, rotated rx 180 ry 0 rz -180 deg; joints [0, 0, 0, 0, 0, 0]
  MoveL (T8306) to (114.56, 103.66, 10.3) mm, rotated rx 180 ry 0 rz -180 deg; joints [0, 0, 0, 0, 0, 0]
  Set speed (40.0 mm/s)
  Call Extruder 2.0
  MoveL (T8307) to (114.56, 103.66, 10.3) mm, rotated rx 180 ry 0 rz -180 deg; joints [0, 0, 0, 0, 0, 0]
  Set speed (26.7 mm/s)
  MoveL (T8308) to (114.56, 103.66, 10.3) mm, rotated rx 180 ry 0 rz -180 deg; joints [0, 0, 0, 0, 0, 0]
  Call Extruder 0.01001
  MoveL (T8309) to (114.75, 103.86, 10.3) mm, rotated rx 180 ry 0 rz -180 deg; joints [0, 0, 0, 0, 0, 0]
  Call Extruder 0.02527
  MoveL (T8310) to (114.75, 104.55, 10.3) mm, rotated rx 180 ry 0 rz -180 deg; joints [0, 0, 0, 0, 0, 0]
  Call Extruder 0.02525
  MoveL (T8311) to (114.27, 104.06, 10.3) mm, rotated rx 180 ry 0 rz -180 deg; joints [0, 0, 0, 0, 0, 0]
  Call Extruder 0.02527
  MoveL (T8312) to (114.27, 104.75, 10.3) mm, rotated rx 180 ry 0 rz -180 deg; joints [0, 0, 0, 0, 0, 0]
  Call Extruder 0.02525
  MoveL (T8313) to (114.75, 105.24, 10.3) mm, rotated rx 180 ry 0 rz -180 deg; joints [0, 0, 0, 0, 0, 0]
  Call Extruder 0.0053
  MoveL (T8314) to (114.76, 105.38, 10.3) mm, rotated rx 180 ry 0 rz -180 deg; joints [0, 0, 0, 0, 0, 0]
  Call Extruder 0.00419
  MoveL (T8315) to (114.67, 105.46, 10.3) mm, rotated rx 180 ry 0 rz -180 deg; joints [0, 0, 0, 0, 0, 0]
  Call Extruder 0.01403
  MoveL (T8316) to (114.29, 105.46, 10.3) mm, rotated rx 180 ry 0 rz -180 deg; joints [0, 0, 0, 0, 0, 0]
  Call Extruder 0.01068
  MoveL (T8317) to (114.08, 105.26, 10.3) mm, rotated rx 180 ry 0 rz -180 deg; joints [0, 0, 0, 0, 0, 0]
  Set speed (45.0 mm/s)
  Call Extruder -1.6
  MoveL (T8318) to (114.08, 105.26, 10.3) mm, rotated rx 180 ry 0 rz -180 deg; joints [0, 0, 0, 0, 0, 0]
  Set speed (120.0 mm/s)
  MoveL (T8319) to (114.08, 105.26, 10.3) mm, rotated rx 180 ry 0 rz -180 deg; joints [0, 0, 0, 0, 0, 0]
  Call Extruder -0.1041
  MoveL (T8320) to (114.29, 105.46, 10.3) mm, rotated rx 180 ry 0 rz -180 deg; joints [0, 0, 0, 0, 0, 0]
  Call Extruder -0.1367
  MoveL (T8321) to (114.67, 105.46, 10.3) mm, rotated rx 180 ry 0 rz -180 deg; joints [0, 0, 0, 0, 0, 0]
  Call Extruder -0.04087
  MoveL (T8322) to (114.76, 105.38, 10.3) mm, rotated rx 180 ry 0 rz -180 deg; joints [0, 0, 0, 0, 0, 0]
  Call Extruder -0.05164
  MoveL (T8323) to (114.75, 105.24, 10.3) mm, rotated rx 180 ry 0 rz -180 deg; joints [0, 0, 0, 0, 0, 0]
  Call Extruder -0.04669
  MoveL (T8324) to (114.66, 105.14, 10.3) mm, rotated rx 180 ry 0 rz -180 deg; joints [0, 0, 0, 0, 0, 0]
  Set speed (45.0 mm/s)
  Call Extruder -0.02
  MoveL (T8325) to (114.66, 105.14, 10.3) mm, rotated rx 180 ry 0 rz -180 deg; joints [0, 0, 0, 0, 0, 0]
  Set speed (150.0 mm/s)
  MoveL (T8326) to (114.66, 105.14, 12.3) mm, rotated rx 180 ry 0 rz -180 deg; joints [0, 0, 0, 0, 0, 0]
  MoveL (T8327) to (116.22, 103.84, 12.3) mm, rotated rx 180 ry 0 rz -180 deg; joints [0, 0, 0, 0, 0, 0]
  MoveL (T8328) to (116.22, 103.84, 10.3) mm, rotated rx 180 ry 0 rz -180 deg; joints [0, 0, 0, 0, 0, 0]
  Set speed (40.0 mm/s)
  Call Extruder 2.0
  MoveL (T8329) to (116.22, 103.84, 10.3) mm, rotated rx 180 ry 0 rz -180 deg; joints [0, 0, 0, 0, 0, 0]
  Set speed (26.7 mm/s)
  MoveL (T8330) to (116.22, 103.84, 10.3) mm, rotated rx 180 ry 0 rz -180 deg; joints [0, 0, 0, 0, 0, 0]
  Call Extruder 0.03214
  MoveL (T8331) to (115.16, 103.84, 10.3) mm, rotated rx 180 ry 0 rz -180 deg; joints [0, 0, 0, 0, 0, 0]
  Call Extruder 0.04227
  MoveL (T8332) to (115.16, 105.23, 10.3) mm, rotated rx 180 ry 0 rz -180 deg; joints [0, 0, 0, 0, 0, 0]
  Call Extruder 0.05977
  MoveL (T8333) to (116.55, 103.84, 10.3) mm, rotated rx 180 ry 0 rz -180 deg; joints [0, 0, 0, 0, 0, 0]
  Call Extruder 0.03385
  MoveL (T8334) to (117.66, 103.84, 10.3) mm, rotated rx 180 ry 0 rz -180 deg; joints [0, 0, 0, 0, 0, 0]
  Call Extruder 0.15054
  MoveL (T8335) to (121.16, 107.34, 10.3) mm, rotated rx 180 ry 0 rz -180 deg; joints [0, 0, 0, 0, 0, 0]
  Call Extruder 0.03385
  MoveL (T8336) to (121.16, 108.45, 10.3) mm, rotated rx 180 ry 0 rz -180 deg; joints [0, 0, 0, 0, 0, 0]
  Call Extruder 0.0017
  MoveL (T8337) to (121.12, 108.49, 10.3) mm, rotated rx 180 ry 0 rz -180 deg; joints [0, 0, 0, 0, 0, 0]
  Call Extruder 0.05185
  MoveL (T8338) to (119.41, 108.49, 10.3) mm, rotated rx 180 ry 0 rz -180 deg; joints [0, 0, 0, 0, 0, 0]
  Call Extruder 0.01373
  MoveL (T8339) to (119.09, 108.81, 10.3) mm, rotated rx 180 ry 0 rz -180 deg; joints [0, 0, 0, 0, 0, 0]
  Call Extruder 0.00882
  MoveL (T8340) to (119.09, 109.1, 10.3) mm, rotated rx 180 ry 0 rz -180 deg; joints [0, 0, 0, 0, 0, 0]
  Set speed (45.0 mm/s)
  Call Extruder -1.6
  MoveL (T8341) to (119.09, 109.1, 10.3) mm, rotated rx 180 ry 0 rz -180 deg; joints [0, 0, 0, 0, 0, 0]
  Set speed (120.0 mm/s)
  MoveL (T8342) to (119.09, 109.1, 10.3) mm, rotated rx 180 ry 0 rz -180 deg; joints [0, 0, 0, 0, 0, 0]
  Call Extruder -0.10318
  MoveL (T8343) to (119.09, 108.81, 10.3) mm, rotated rx 180 ry 0 rz -180 deg; joints [0, 0, 0, 0, 0, 0]
  Call Extruder -0.16059
  MoveL (T8344) to (119.41, 108.49, 10.3) mm, rotated rx 180 ry 0 rz -180 deg; joints [0, 0, 0, 0, 0, 0]
  Call Extruder -0.11623
  MoveL (T8345) to (119.74, 108.49, 10.3) mm, rotated rx 180 ry 0 rz -180 deg; joints [0, 0, 0, 0, 0, 0]
  Set speed (45.0 mm/s)
  Call Extruder -0.02
  MoveL (T8346) to (119.74, 108.49, 10.3) mm, rotated rx 180 ry 0 rz -180 deg; joints [0, 0, 0, 0, 0, 0]
  Set speed (150.0 mm/s)
  MoveL (T8347) to (119.74, 108.49, 12.3) mm, rotated rx 180 ry 0 rz -180 deg; joints [0, 0, 0, 0, 0, 0]
  MoveL (T8348) to (121.34, 109.09, 12.3) mm, rotated rx 180 ry 0 rz -180 deg; joints [0, 0, 0, 0, 0, 0]
  MoveL (T8349) to (121.34, 109.09, 10.3) mm, rotated rx 180 ry 0 rz -180 deg; joints [0, 0, 0, 0, 0, 0]
  Set speed (40.0 mm/s)
  Call Extruder 2.0
  MoveL (T8350) to (121.34, 109.09, 10.3) mm, rotated rx 180 ry 0 rz -180 deg; joints [0, 0, 0, 0, 0, 0]
  Set speed (26.7 mm/s)
  MoveL (T8351) to (121.34, 109.09, 10.3) mm, rotated rx 180 ry 0 rz -180 deg; joints [0, 0, 0, 0, 0, 0]
  Call Extruder 0.01001
  MoveL (T8352) to (121.14, 108.9, 10.3) mm, rotated rx 180 ry 0 rz -180 deg; joints [0, 0, 0, 0, 0, 0]
  Call Extruder 0.02524
  MoveL (T8353) to (120.45, 108.9, 10.3) mm, rotated rx 180 ry 0 rz -180 deg; joints [0, 0, 0, 0, 0, 0]
  Call Extruder 0.02268
  MoveL (T8354) to (120.89, 109.34, 10.3) mm, rotated rx 180 ry 0 rz -180 deg; joints [0, 0, 0, 0, 0, 0]
  Call Extruder 0.02524
  MoveL (T8355) to (120.2, 109.34, 10.3) mm, rotated rx 180 ry 0 rz -180 deg; joints [0, 0, 0, 0, 0, 0]
  Call Extruder 0.02268
  MoveL (T8356) to (119.76, 108.9, 10.3) mm, rotated rx 180 ry 0 rz -180 deg; joints [0, 0, 0, 0, 0, 0]
  Call Extruder 0.00664
  MoveL (T8357) to (119.58, 108.9, 10.3) mm, rotated rx 180 ry 0 rz -180 deg; joints [0, 0, 0, 0, 0, 0]
  Call Extruder 0.00418
  MoveL (T8358) to (119.5, 108.98, 10.3) mm, rotated rx 180 ry 0 rz -180 deg; joints [0, 0, 0, 0, 0, 0]
  Call Extruder 0.01266
  MoveL (T8359) to (119.5, 109.32, 10.3) mm, rotated rx 180 ry 0 rz -180 deg; joints [0, 0, 0, 0, 0, 0]
  Call Extruder 0.01008
  MoveL (T8360) to (119.69, 109.52, 10.3) mm, rotated rx 180 ry 0 rz -180 deg; joints [0, 0, 0, 0, 0, 0]
  Set speed (45.0 mm/s)
  Call Extruder -1.6
  MoveL (T8361) to (119.69, 109.52, 10.3) mm, rotated rx 180 ry 0 rz -180 deg; joints [0, 0, 0, 0, 0, 0]
  Set speed (120.0 mm/s)
  MoveL (T8362) to (119.69, 109.52, 10.3) mm, rotated rx 180 ry 0 rz -180 deg; joints [0, 0, 0, 0, 0, 0]
  Call Extruder -0.09819
  MoveL (T8363) to (119.5, 109.32, 10.3) mm, rotated rx 180 ry 0 rz -180 deg; joints [0, 0, 0, 0, 0, 0]
  Call Extruder -0.12336
  MoveL (T8364) to (119.5, 108.98, 10.3) mm, rotated rx 180 ry 0 rz -180 deg; joints [0, 0, 0, 0, 0, 0]
  Call Extruder -0.04075
  MoveL (T8365) to (119.58, 108.9, 10.3) mm, rotated rx 180 ry 0 rz -180 deg; joints [0, 0, 0, 0, 0, 0]
  Call Extruder -0.06472
  MoveL (T8366) to (119.76, 108.9, 10.3) mm, rotated rx 180 ry 0 rz -180 deg; joints [0, 0, 0, 0, 0, 0]
  Call Extruder -0.05298
  MoveL (T8367) to (119.87, 109, 10.3) mm, rotated rx 180 ry 0 rz -180 deg; joints [0, 0, 0, 0, 0, 0]
  Set speed (45.0 mm/s)
  Call Extruder -0.02
  MoveL (T8368) to (119.87, 109, 10.3) mm, rotated rx 180 ry 0 rz -180 deg; joints [0, 0, 0, 0, 0, 0]
  Set speed (150.0 mm/s)
  MoveL (T8369) to (119.87, 109, 12.3) mm, rotated rx 180 ry 0 rz -180 deg; joints [0, 0, 0, 0, 0, 0]
  MoveL (T8370) to (118.71, 103.84, 12.3) mm, rotated rx 180 ry 0 rz -180 deg; joints [0, 0, 0, 0, 0, 0]
  MoveL (T8371) to (118.71, 103.84, 10.3) mm, rotated rx 180 ry 0 rz -180 deg; joints [0, 0, 0, 0, 0, 0]
  Set speed (40.0 mm/s)
  Call Extruder 2.0
  MoveL (T8372) to (118.71, 103.84, 10.3) mm, rotated rx 180 ry 0 rz -180 deg; joints [0, 0, 0, 0, 0, 0]
  Set speed (26.7 mm/s)
  MoveL (T8373) to (118.71, 103.84, 10.3) mm, rotated rx 180 ry 0 rz -180 deg; joints [0, 0, 0, 0, 0, 0]
  Call Extruder 0.07441
  MoveL (T8374) to (121.16, 103.84, 10.3) mm, rotated rx 180 ry 0 rz -180 deg; joints [0, 0, 0, 0, 0, 0]
  Call Extruder 0.7458
  MoveL (T8375) to (103.84, 121.16, 10.3) mm, rotated rx 180 ry 0 rz -180 deg; joints [0, 0, 0, 0, 0, 0]
  Call Extruder 0.10645
  MoveL (T8376) to (103.84, 117.66, 10.3) mm, rotated rx 180 ry 0 rz -180 deg; joints [0, 0, 0, 0, 0, 0]
  Call Extruder 0.15054
  MoveL (T8377) to (107.34, 121.16, 10.3) mm, rotated rx 180 ry 0 rz -180 deg; joints [0, 0, 0, 0, 0, 0]
  Call Extruder 0.03385
  MoveL (T8378) to (108.45, 121.16, 10.3) mm, rotated rx 180 ry 0 rz -180 deg; joints [0, 0, 0, 0, 0, 0]
  Call Extruder 0.46402
  MoveL (T8379) to (119.22, 110.39, 10.3) mm, rotated rx 180 ry 0 rz -180 deg; joints [0, 0, 0, 0, 0, 0]
  Call Extruder 0.01144
  MoveL (T8380) to (119.22, 110.01, 10.3) mm, rotated rx 180 ry 0 rz -180 deg; joints [0, 0, 0, 0, 0, 0]
  Call Extruder 0.18346
  MoveL (T8381) to (114.96, 105.75, 10.3) mm, rotated rx 180 ry 0 rz -180 deg; joints [0, 0, 0, 0, 0, 0]
  Call Extruder 0.00514
  MoveL (T8382) to (114.84, 105.87, 10.3) mm, rotated rx 180 ry 0 rz -180 deg; joints [0, 0, 0, 0, 0, 0]
  Call Extruder 0.00972
  MoveL (T8383) to (114.52, 105.87, 10.3) mm, rotated rx 180 ry 0 rz -180 deg; joints [0, 0, 0, 0, 0, 0]
  Call Extruder 0.4601
  MoveL (T8384) to (103.84, 116.55, 10.3) mm, rotated rx 180 ry 0 rz -180 deg; joints [0, 0, 0, 0, 0, 0]
  Call Extruder 0.10645
  MoveL (T8385) to (103.84, 113.06, 10.3) mm, rotated rx 180 ry 0 rz -180 deg; joints [0, 0, 0, 0, 0, 0]
  Call Extruder 0.34896
  MoveL (T8386) to (111.94, 121.16, 10.3) mm, rotated rx 180 ry 0 rz -180 deg; joints [0, 0, 0, 0, 0, 0]
  Call Extruder 0.03385
  MoveL (T8387) to (113.06, 121.16, 10.3) mm, rotated rx 180 ry 0 rz -180 deg; joints [0, 0, 0, 0, 0, 0]
  Call Extruder 0.26005
  MoveL (T8388) to (119.09, 115.12, 10.3) mm, rotated rx 180 ry 0 rz -180 deg; joints [0, 0, 0, 0, 0, 0]
  Call Extruder 0.01502
  MoveL (T8389) to (119.09, 114.63, 10.3) mm, rotated rx 180 ry 0 rz -180 deg; joints [0, 0, 0, 0, 0, 0]
  Call Extruder 0.00304
  MoveL (T8390) to (119.16, 114.56, 10.3) mm, rotated rx 180 ry 0 rz -180 deg; joints [0, 0, 0, 0, 0, 0]
  Call Extruder 0.37974
  MoveL (T8391) to (110.35, 105.74, 10.3) mm, rotated rx 180 ry 0 rz -180 deg; joints [0, 0, 0, 0, 0, 0]
  Call Extruder 0.00912
  MoveL (T8392) to (110.05, 105.74, 10.3) mm, rotated rx 180 ry 0 rz -180 deg; joints [0, 0, 0, 0, 0, 0]
  Call Extruder 0.26725
  MoveL (T8393) to (103.84, 111.94, 10.3) mm, rotated rx 180 ry 0 rz -180 deg; joints [0, 0, 0, 0, 0, 0]
  Call Extruder 0.07441
  MoveL (T8394) to (103.84, 109.5, 10.3) mm, rotated rx 180 ry 0 rz -180 deg; joints [0, 0, 0, 0, 0, 0]
  Set speed (45.0 mm/s)
  Call Extruder -1.6
  MoveL (T8395) to (103.84, 109.5, 10.3) mm, rotated rx 180 ry 0 rz -180 deg; joints [0, 0, 0, 0, 0, 0]
  Set speed (120.0 mm/s)
  MoveL (T8396) to (103.84, 109.5, 10.3) mm, rotated rx 180 ry 0 rz -180 deg; joints [0, 0, 0, 0, 0, 0]
  Call Extruder -0.38
  MoveL (T8397) to (103.84, 110.57, 10.3) mm, rotated rx 180 ry 0 rz -180 deg; joints [0, 0, 0, 0, 0, 0]
  Set speed (45.0 mm/s)
  Call Extruder -0.02
  MoveL (T8398) to (103.84, 110.57, 10.3) mm, rotated rx 180 ry 0 rz -180 deg; joints [0, 0, 0, 0, 0, 0]
  Set speed (150.0 mm/s)
  MoveL (T8399) to (103.84, 110.57, 12.3) mm, rotated rx 180 ry 0 rz -180 deg; joints [0, 0, 0, 0, 0, 0]
  MoveL (T8400) to (121.14, 115.43, 12.3) mm, rotated rx 180 ry 0 rz -180 deg; joints [0, 0, 0, 0, 0, 0]
  MoveL (T8401) to (121.14, 115.43, 10.3) mm, rotated rx 180 ry 0 rz -180 deg; joints [0, 0, 0, 0, 0, 0]
  Set speed (40.0 mm/s)
  Call Extruder 2.0
  MoveL (T8402) to (121.14, 115.43, 10.3) mm, rotated rx 180 ry 0 rz -180 deg; joints [0, 0, 0, 0, 0, 0]
  Set speed (26.7 mm/s)
  MoveL (T8403) to (121.14, 115.43, 10.3) mm, rotated rx 180 ry 0 rz -180 deg; joints [0, 0, 0, 0, 0, 0]
  Call Extruder 0.02922
  MoveL (T8404) to (120.56, 114.84, 10.3) mm, rotated rx 180 ry 0 rz -180 deg; joints [0, 0, 0, 0, 0, 0]
  Call Extruder 0.0236
  MoveL (T8405) to (119.89, 114.84, 10.3) mm, rotated rx 180 ry 0 rz -180 deg; joints [0, 0, 0, 0, 0, 0]
  Call Extruder 0.02006
  MoveL (T8406) to (120.29, 115.24, 10.3) mm, rotated rx 180 ry 0 rz -180 deg; joints [0, 0, 0, 0, 0, 0]
  Call Extruder 0.0236
  MoveL (T8407) to (119.63, 115.24, 10.3) mm, rotated rx 180 ry 0 rz -180 deg; joints [0, 0, 0, 0, 0, 0]
  Call Extruder 0.0155
  MoveL (T8408) to (119.31, 114.93, 10.3) mm, rotated rx 180 ry 0 rz -180 deg; joints [0, 0, 0, 0, 0, 0]
  Set speed (45.0 mm/s)
  Call Extruder -1.6
  MoveL (T8409) to (119.31, 114.93, 10.3) mm, rotated rx 180 ry 0 rz -180 deg; joints [0, 0, 0, 0, 0, 0]
  Set speed (120.0 mm/s)
  MoveL (T8410) to (119.31, 114.93, 10.3) mm, rotated rx 180 ry 0 rz -180 deg; joints [0, 0, 0, 0, 0, 0]
  Call Extruder -0.15634
  MoveL (T8411) to (119.63, 115.24, 10.3) mm, rotated rx 180 ry 0 rz -180 deg; joints [0, 0, 0, 0, 0, 0]
  Call Extruder -0.22366
  MoveL (T8412) to (120.25, 115.24, 10.3) mm, rotated rx 180 ry 0 rz -180 deg; joints [0, 0, 0, 0, 0, 0]
  Set speed (45.0 mm/s)
  Call Extruder -0.02
  MoveL (T8413) to (120.25, 115.24, 10.3) mm, rotated rx 180 ry 0 rz -180 deg; joints [0, 0, 0, 0, 0, 0]
  Set speed (150.0 mm/s)
  MoveL (T8414) to (120.25, 115.24, 12.3) mm, rotated rx 180 ry 0 rz -180 deg; joints [0, 0, 0, 0, 0, 0]
  MoveL (T8415) to (104.34, 103.54, 12.3) mm, rotated rx 180 ry 0 rz -180 deg; joints [0, 0, 0, 0, 0, 0]
  MoveL (T8416) to (104.34, 103.54, 10.5) mm, rotated rx 180 ry 0 rz -180 deg; joints [0, 0, 0, 0, 0, 0]
  Set speed (40.0 mm/s)
  Call Extruder 2.0
  MoveL (T8417) to (104.34, 103.54, 10.5) mm, rotated rx 180 ry 0 rz -180 deg; joints [0, 0, 0, 0, 0, 0]
  Set speed (24.9 mm/s)
  MoveL (T8418) to (104.34, 103.54, 10.5) mm, rotated rx 180 ry 0 rz -180 deg; joints [0, 0, 0, 0, 0, 0]
  Call Extruder 0.16816
  MoveL (T8419) to (109.86, 103.54, 10.5) mm, rotated rx 180 ry 0 rz -180 deg; joints [0, 0, 0, 0, 0, 0]
  Call Extruder 0.05779
  MoveL (T8420) to (109.86, 105.44, 10.5) mm, rotated rx 180 ry 0 rz -180 deg; joints [0, 0, 0, 0, 0, 0]
  Call Extruder 0.12892
  MoveL (T8421) to (114.09, 105.44, 10.5) mm, rotated rx 180 ry 0 rz -180 deg; joints [0, 0, 0, 0, 0, 0]
  Call Extruder 0.05779
  MoveL (T8422) to (114.09, 103.54, 10.5) mm, rotated rx 180 ry 0 rz -180 deg; joints [0, 0, 0, 0, 0, 0]
  Call Extruder 0.22458
  MoveL (T8423) to (121.46, 103.54, 10.5) mm, rotated rx 180 ry 0 rz -180 deg; joints [0, 0, 0, 0, 0, 0]
  Call Extruder 0.18223
  MoveL (T8424) to (121.46, 109.52, 10.5) mm, rotated rx 180 ry 0 rz -180 deg; joints [0, 0, 0, 0, 0, 0]
  Call Extruder 0.05893
  MoveL (T8425) to (119.53, 109.52, 10.5) mm, rotated rx 180 ry 0 rz -180 deg; joints [0, 0, 0, 0, 0, 0]
  Call Extruder 0.1562
  MoveL (T8426) to (119.52, 114.65, 10.5) mm, rotated rx 180 ry 0 rz -180 deg; joints [0, 0, 0, 0, 0, 0]
  Call Extruder 0.059
  MoveL (T8427) to (121.46, 114.65, 10.5) mm, rotated rx 180 ry 0 rz -180 deg; joints [0, 0, 0, 0, 0, 0]
  Call Extruder 0.20743
  MoveL (T8428) to (121.46, 121.46, 10.5) mm, rotated rx 180 ry 0 rz -180 deg; joints [0, 0, 0, 0, 0, 0]
  Call Extruder 0.54596
  MoveL (T8429) to (103.54, 121.46, 10.5) mm, rotated rx 180 ry 0 rz -180 deg; joints [0, 0, 0, 0, 0, 0]
  Call Extruder 0.54596
  MoveL (T8430) to (103.54, 103.54, 10.5) mm, rotated rx 180 ry 0 rz -180 deg; joints [0, 0, 0, 0, 0, 0]
  Call Extruder 0.02254
  MoveL (T8431) to (104.28, 103.54, 10.5) mm, rotated rx 180 ry 0 rz -180 deg; joints [0, 0, 0, 0, 0, 0]
  Set speed (150.0 mm/s)
  MoveL (T8432) to (103.53, 103.13, 10.5) mm, rotated rx 180 ry 0 rz -180 deg; joints [0, 0, 0, 0, 0, 0]
  Set speed (24.9 mm/s)
  MoveL (T8433) to (103.53, 103.13, 10.5) mm, rotated rx 180 ry 0 rz -180 deg; joints [0, 0, 0, 0, 0, 0]
  Call Extruder 0.20515
  MoveL (T8434) to (110.27, 103.13, 10.5) mm, rotated rx 180 ry 0 rz -180 deg; joints [0, 0, 0, 0, 0, 0]
  Call Extruder 0.05779
  MoveL (T8435) to (110.27, 105.03, 10.5) mm, rotated rx 180 ry 0 rz -180 deg; joints [0, 0, 0, 0, 0, 0]
  Call Extruder 0.1041
  MoveL (T8436) to (113.68, 105.03, 10.5) mm, rotated rx 180 ry 0 rz -180 deg; joints [0, 0, 0, 0, 0, 0]
  Call Extruder 0.05779
  MoveL (T8437) to (113.68, 103.13, 10.5) mm, rotated rx 180 ry 0 rz -180 deg; joints [0, 0, 0, 0, 0, 0]
  Call Extruder 0.24939
  MoveL (T8438) to (121.87, 103.13, 10.5) mm, rotated rx 180 ry 0 rz -180 deg; joints [0, 0, 0, 0, 0, 0]
  Call Extruder 0.20703
  MoveL (T8439) to (121.87, 109.93, 10.5) mm, rotated rx 180 ry 0 rz -180 deg; joints [0, 0, 0, 0, 0, 0]
  Call Extruder 0.05893
  MoveL (T8440) to (119.93, 109.93, 10.5) mm, rotated rx 180 ry 0 rz -180 deg; joints [0, 0, 0, 0, 0, 0]
  Call Extruder 0.13142
  MoveL (T8441) to (119.93, 114.24, 10.5) mm, rotated rx 180 ry 0 rz -180 deg; joints [0, 0, 0, 0, 0, 0]
  Call Extruder 0.05899
  MoveL (T8442) to (121.87, 114.25, 10.5) mm, rotated rx 180 ry 0 rz -180 deg; joints [0, 0, 0, 0, 0, 0]
  Call Extruder 0.23222
  MoveL (T8443) to (121.87, 121.87, 10.5) mm, rotated rx 180 ry 0 rz -180 deg; joints [0, 0, 0, 0, 0, 0]
  Call Extruder 0.57077
  MoveL (T8444) to (103.13, 121.87, 10.5) mm, rotated rx 180 ry 0 rz -180 deg; joints [0, 0, 0, 0, 0, 0]
  Call Extruder 0.57077
  MoveL (T8445) to (103.13, 103.13, 10.5) mm, rotated rx 180 ry 0 rz -180 deg; joints [0, 0, 0, 0, 0, 0]
  Call Extruder 0.01036
  MoveL (T8446) to (103.47, 103.13, 10.5) mm, rotated rx 180 ry 0 rz -180 deg; joints [0, 0, 0, 0, 0, 0]
  Set speed (150.0 mm/s)
  MoveL (T8447) to (102.72, 102.81, 10.5) mm, rotated rx 180 ry 0 rz -180 deg; joints [0, 0, 0, 0, 0, 0]
  Set speed (24.9 mm/s)
  MoveL (T8448) to (102.72, 102.81, 10.5) mm, rotated rx 180 ry 0 rz -180 deg; joints [0, 0, 0, 0, 0, 0]
  Call Extruder 0.00259
  MoveL (T8449) to (102.72, 102.72, 10.5) mm, rotated rx 180 ry 0 rz -180 deg; joints [0, 0, 0, 0, 0, 0]
  Call Extruder 0.24214
  MoveL (T8450) to (110.67, 102.72, 10.5) mm, rotated rx 180 ry 0 rz -180 deg; joints [0, 0, 0, 0, 0, 0]
  Call Extruder 0.05779
  MoveL (T8451) to (110.67, 104.62, 10.5) mm, rotated rx 180 ry 0 rz -180 deg; joints [0, 0, 0, 0, 0, 0]
  Call Extruder 0.07929
  MoveL (T8452) to (113.28, 104.62, 10.5) mm, rotated rx 180 ry 0 rz -180 deg; joints [0, 0, 0, 0, 0, 0]
  Call Extruder 0.05779
  MoveL (T8453) to (113.27, 102.72, 10.5) mm, rotated rx 180 ry 0 rz -180 deg; joints [0, 0, 0, 0, 0, 0]
  Call Extruder 0.2742
  MoveL (T8454) to (122.28, 102.72, 10.5) mm, rotated rx 180 ry 0 rz -180 deg; joints [0, 0, 0, 0, 0, 0]
  Call Extruder 0.23182
  MoveL (T8455) to (122.28, 110.33, 10.5) mm, rotated rx 180 ry 0 rz -180 deg; joints [0, 0, 0, 0, 0, 0]
  Call Extruder 0.05894
  MoveL (T8456) to (120.34, 110.34, 10.5) mm, rotated rx 180 ry 0 rz -180 deg; joints [0, 0, 0, 0, 0, 0]
  Call Extruder 0.10664
  MoveL (T8457) to (120.34, 113.84, 10.5) mm, rotated rx 180 ry 0 rz -180 deg; joints [0, 0, 0, 0, 0, 0]
  Call Extruder 0.05899
  MoveL (T8458) to (122.28, 113.84, 10.5) mm, rotated rx 180 ry 0 rz -180 deg; joints [0, 0, 0, 0, 0, 0]
  Call Extruder 0.25701
  MoveL (T8459) to (122.28, 122.28, 10.5) mm, rotated rx 180 ry 0 rz -180 deg; joints [0, 0, 0, 0, 0, 0]
  Call Extruder 0.59557
  MoveL (T8460) to (102.72, 122.28, 10.5) mm, rotated rx 180 ry 0 rz -180 deg; joints [0, 0, 0, 0, 0, 0]
  Call Extruder 0.59115
  MoveL (T8461) to (102.72, 102.87, 10.5) mm, rotated rx 180 ry 0 rz -180 deg; joints [0, 0, 0, 0, 0, 0]
  Set speed (150.0 mm/s)
  MoveL (T8462) to (102.78, 102.75, 10.5) mm, rotated rx 180 ry 0 rz -180 deg; joints [0, 0, 0, 0, 0, 0]
  Set speed (45.0 mm/s)
  Call Extruder -1.6
  MoveL (T8463) to (102.78, 102.75, 10.5) mm, rotated rx 180 ry 0 rz -180 deg; joints [0, 0, 0, 0, 0, 0]
  Set speed (120.0 mm/s)
  MoveL (T8464) to (102.78, 102.75, 10.5) mm, rotated rx 180 ry 0 rz -180 deg; joints [0, 0, 0, 0, 0, 0]
  Call Extruder -0.05166
  MoveL (T8465) to (102.72, 102.72, 10.5) mm, rotated rx 180 ry 0 rz -180 deg; joints [0, 0, 0, 0, 0, 0]
  Call Extruder -0.32834
  MoveL (T8466) to (103.65, 102.72, 10.5) mm, rotated rx 180 ry 0 rz -180 deg; joints [0, 0, 0, 0, 0, 0]
  Set speed (45.0 mm/s)
  Call Extruder -0.02
  MoveL (T8467) to (103.65, 102.72, 10.5) mm, rotated rx 180 ry 0 rz -180 deg; joints [0, 0, 0, 0, 0, 0]
  Set speed (150.0 mm/s)
  MoveL (T8468) to (103.65, 102.72, 12.5) mm, rotated rx 180 ry 0 rz -180 deg; joints [0, 0, 0, 0, 0, 0]
  MoveL (T8469) to (106.29, 103.84, 12.5) mm, rotated rx 180 ry 0 rz -180 deg; joints [0, 0, 0, 0, 0, 0]
  MoveL (T8470) to (106.29, 103.84, 10.5) mm, rotated rx 180 ry 0 rz -180 deg; joints [0, 0, 0, 0, 0, 0]
  Set speed (40.0 mm/s)
  Call Extruder 2.0
  MoveL (T8471) to (106.29, 103.84, 10.5) mm, rotated rx 180 ry 0 rz -180 deg; joints [0, 0, 0, 0, 0, 0]
  Set speed (24.9 mm/s)
  MoveL (T8472) to (106.29, 103.84, 10.5) mm, rotated rx 180 ry 0 rz -180 deg; joints [0, 0, 0, 0, 0, 0]
  Call Extruder 0.07441
  MoveL (T8473) to (103.84, 103.84, 10.5) mm, rotated rx 180 ry 0 rz -180 deg; joints [0, 0, 0, 0, 0, 0]
  Call Extruder 0.7458
  MoveL (T8474) to (121.16, 121.16, 10.5) mm, rotated rx 180 ry 0 rz -180 deg; joints [0, 0, 0, 0, 0, 0]
  Call Extruder 0.07441
  MoveL (T8475) to (118.71, 121.16, 10.5) mm, rotated rx 180 ry 0 rz -180 deg; joints [0, 0, 0, 0, 0, 0]
  Set speed (45.0 mm/s)
  Call Extruder -1.6
  MoveL (T8476) to (118.71, 121.16, 10.5) mm, rotated rx 180 ry 0 rz -180 deg; joints [0, 0, 0, 0, 0, 0]
  Set speed (120.0 mm/s)
  MoveL (T8477) to (118.71, 121.16, 10.5) mm, rotated rx 180 ry 0 rz -180 deg; joints [0, 0, 0, 0, 0, 0]
  Call Extruder -0.38
  MoveL (T8478) to (119.78, 121.16, 10.5) mm, rotated rx 180 ry 0 rz -180 deg; joints [0, 0, 0, 0, 0, 0]
  Set speed (45.0 mm/s)
  Call Extruder -0.02
  MoveL (T8479) to (119.78, 121.16, 10.5) mm, rotated rx 180 ry 0 rz -180 deg; joints [0, 0, 0, 0, 0, 0]
  Set speed (150.0 mm/s)
  MoveL (T8480) to (119.78, 121.16, 12.5) mm, rotated rx 180 ry 0 rz -180 deg; joints [0, 0, 0, 0, 0, 0]
  MoveL (T8481) to (121.17, 108.59, 12.5) mm, rotated rx 180 ry 0 rz -180 deg; joints [0, 0, 0, 0, 0, 0]
  MoveL (T8482) to (121.17, 108.59, 10.5) mm, rotated rx 180 ry 0 rz -180 deg; joints [0, 0, 0, 0, 0, 0]
  Set speed (40.0 mm/s)
  Call Extruder 2.0
  MoveL (T8483) to (121.17, 108.59, 10.5) mm, rotated rx 180 ry 0 rz -180 deg; joints [0, 0, 0, 0, 0, 0]
  Set speed (24.9 mm/s)
  MoveL (T8484) to (121.17, 108.59, 10.5) mm, rotated rx 180 ry 0 rz -180 deg; joints [0, 0, 0, 0, 0, 0]
  Call Extruder 0.03151
  MoveL (T8485) to (120.55, 109.22, 10.5) mm, rotated rx 180 ry 0 rz -180 deg; joints [0, 0, 0, 0, 0, 0]
  Call Extruder 0.02423
  MoveL (T8486) to (119.87, 109.22, 10.5) mm, rotated rx 180 ry 0 rz -180 deg; joints [0, 0, 0, 0, 0, 0]
  Call Extruder 0.02223
  MoveL (T8487) to (120.31, 108.78, 10.5) mm, rotated rx 180 ry 0 rz -180 deg; joints [0, 0, 0, 0, 0, 0]
  Call Extruder 0.02423
  MoveL (T8488) to (119.63, 108.78, 10.5) mm, rotated rx 180 ry 0 rz -180 deg; joints [0, 0, 0, 0, 0, 0]
  Call Extruder 0.01594
  MoveL (T8489) to (119.32, 109.09, 10.5) mm, rotated rx 180 ry 0 rz -180 deg; joints [0, 0, 0, 0, 0, 0]
  Set speed (45.0 mm/s)
  Call Extruder -1.6
  MoveL (T8490) to (119.32, 109.09, 10.5) mm, rotated rx 180 ry 0 rz -180 deg; joints [0, 0, 0, 0, 0, 0]
  Set speed (120.0 mm/s)
  MoveL (T8491) to (119.32, 109.09, 10.5) mm, rotated rx 180 ry 0 rz -180 deg; joints [0, 0, 0, 0, 0, 0]
  Call Extruder -0.15865
  MoveL (T8492) to (119.63, 108.78, 10.5) mm, rotated rx 180 ry 0 rz -180 deg; joints [0, 0, 0, 0, 0, 0]
  Call Extruder -0.22135
  MoveL (T8493) to (120.25, 108.78, 10.5) mm, rotated rx 180 ry 0 rz -180 deg; joints [0, 0, 0, 0, 0, 0]
  Set speed (45.0 mm/s)
  Call Extruder -0.02
  MoveL (T8494) to (120.25, 108.78, 10.5) mm, rotated rx 180 ry 0 rz -180 deg; joints [0, 0, 0, 0, 0, 0]
  Set speed (150.0 mm/s)
  MoveL (T8495) to (120.25, 108.78, 12.5) mm, rotated rx 180 ry 0 rz -180 deg; joints [0, 0, 0, 0, 0, 0]
  MoveL (T8496) to (121.34, 115.17, 12.5) mm, rotated rx 180 ry 0 rz -180 deg; joints [0, 0, 0, 0, 0, 0]
  MoveL (T8497) to (121.34, 115.17, 10.5) mm, rotated rx 180 ry 0 rz -180 deg; joints [0, 0, 0, 0, 0, 0]
  Set speed (40.0 mm/s)
  Call Extruder 2.0
  MoveL (T8498) to (121.34, 115.17, 10.5) mm, rotated rx 180 ry 0 rz -180 deg; joints [0, 0, 0, 0, 0, 0]
  Set speed (24.9 mm/s)
  MoveL (T8499) to (121.34, 115.17, 10.5) mm, rotated rx 180 ry 0 rz -180 deg; joints [0, 0, 0, 0, 0, 0]
  Call Extruder 0.00968
  MoveL (T8500) to (121.15, 115.36, 10.5) mm, rotated rx 180 ry 0 rz -180 deg; joints [0, 0, 0, 0, 0, 0]
  Call Extruder 0.02462
  MoveL (T8501) to (120.47, 115.36, 10.5) mm, rotated rx 180 ry 0 rz -180 deg; joints [0, 0, 0, 0, 0, 0]
  Call Extruder 0.02046
  MoveL (T8502) to (120.87, 114.96, 10.5) mm, rotated rx 180 ry 0 rz -180 deg; joints [0, 0, 0, 0, 0, 0]
  Call Extruder 0.02462
  MoveL (T8503) to (120.19, 114.95, 10.5) mm, rotated rx 180 ry 0 rz -180 deg; joints [0, 0, 0, 0, 0, 0]
  Call Extruder 0.02046
  MoveL (T8504) to (119.79, 115.36, 10.5) mm, rotated rx 180 ry 0 rz -180 deg; joints [0, 0, 0, 0, 0, 0]
  Call Extruder 0.00743
  MoveL (T8505) to (119.58, 115.36, 10.5) mm, rotated rx 180 ry 0 rz -180 deg; joints [0, 0, 0, 0, 0, 0]
  Call Extruder 0.00413
  MoveL (T8506) to (119.5, 115.28, 10.5) mm, rotated rx 180 ry 0 rz -180 deg; joints [0, 0, 0, 0, 0, 0]
  Call Extruder 0.01134
  MoveL (T8507) to (119.5, 114.96, 10.5) mm, rotated rx 180 ry 0 rz -180 deg; joints [0, 0, 0, 0, 0, 0]
  Call Extruder 0.00967
  MoveL (T8508) to (119.69, 114.77, 10.5) mm, rotated rx 180 ry 0 rz -180 deg; joints [0, 0, 0, 0, 0, 0]
  Set speed (150.0 mm/s)
  MoveL (T8509) to (119.09, 115.32, 10.5) mm, rotated rx 180 ry 0 rz -180 deg; joints [0, 0, 0, 0, 0, 0]
  Set speed (24.9 mm/s)
  MoveL (T8510) to (119.09, 115.32, 10.5) mm, rotated rx 180 ry 0 rz -180 deg; joints [0, 0, 0, 0, 0, 0]
  Call Extruder 0.00368
  MoveL (T8511) to (119.09, 115.44, 10.5) mm, rotated rx 180 ry 0 rz -180 deg; joints [0, 0, 0, 0, 0, 0]
  Call Extruder 0.01373
  MoveL (T8512) to (119.41, 115.76, 10.5) mm, rotated rx 180 ry 0 rz -180 deg; joints [0, 0, 0, 0, 0, 0]
  Call Extruder 0.02918
  MoveL (T8513) to (120.37, 115.76, 10.5) mm, rotated rx 180 ry 0 rz -180 deg; joints [0, 0, 0, 0, 0, 0]
  Call Extruder 0.03387
  MoveL (T8514) to (121.16, 116.55, 10.5) mm, rotated rx 180 ry 0 rz -180 deg; joints [0, 0, 0, 0, 0, 0]
  Call Extruder 0.03385
  MoveL (T8515) to (121.16, 117.66, 10.5) mm, rotated rx 180 ry 0 rz -180 deg; joints [0, 0, 0, 0, 0, 0]
  Call Extruder 0.15054
  MoveL (T8516) to (117.66, 121.16, 10.5) mm, rotated rx 180 ry 0 rz -180 deg; joints [0, 0, 0, 0, 0, 0]
  Call Extruder 0.03385
  MoveL (T8517) to (116.55, 121.16, 10.5) mm, rotated rx 180 ry 0 rz -180 deg; joints [0, 0, 0, 0, 0, 0]
  Call Extruder 0.54738
  MoveL (T8518) to (103.84, 108.45, 10.5) mm, rotated rx 180 ry 0 rz -180 deg; joints [0, 0, 0, 0, 0, 0]
  Call Extruder 0.03385
  MoveL (T8519) to (103.84, 107.34, 10.5) mm, rotated rx 180 ry 0 rz -180 deg; joints [0, 0, 0, 0, 0, 0]
  Call Extruder 0.15054
  MoveL (T8520) to (107.34, 103.84, 10.5) mm, rotated rx 180 ry 0 rz -180 deg; joints [0, 0, 0, 0, 0, 0]
  Call Extruder 0.03385
  MoveL (T8521) to (108.45, 103.84, 10.5) mm, rotated rx 180 ry 0 rz -180 deg; joints [0, 0, 0, 0, 0, 0]
  Call Extruder 0.01294
  MoveL (T8522) to (108.75, 104.14, 10.5) mm, rotated rx 180 ry 0 rz -180 deg; joints [0, 0, 0, 0, 0, 0]
  Call Extruder 0.04284
  MoveL (T8523) to (108.75, 105.55, 10.5) mm, rotated rx 180 ry 0 rz -180 deg; joints [0, 0, 0, 0, 0, 0]
  Call Extruder 0.01377
  MoveL (T8524) to (109.07, 105.87, 10.5) mm, rotated rx 180 ry 0 rz -180 deg; joints [0, 0, 0, 0, 0, 0]
  Call Extruder 0.0178
  MoveL (T8525) to (109.65, 105.87, 10.5) mm, rotated rx 180 ry 0 rz -180 deg; joints [0, 0, 0, 0, 0, 0]
  Set speed (150.0 mm/s)
  MoveL (T8526) to (109.74, 105.28, 10.5) mm, rotated rx 180 ry 0 rz -180 deg; joints [0, 0, 0, 0, 0, 0]
  Set speed (24.9 mm/s)
  MoveL (T8527) to (109.74, 105.28, 10.5) mm, rotated rx 180 ry 0 rz -180 deg; joints [0, 0, 0, 0, 0, 0]
  Call Extruder 0.00923
  MoveL (T8528) to (109.55, 105.46, 10.5) mm, rotated rx 180 ry 0 rz -180 deg; joints [0, 0, 0, 0, 0, 0]
  Call Extruder 0.01116
  MoveL (T8529) to (109.24, 105.46, 10.5) mm, rotated rx 180 ry 0 rz -180 deg; joints [0, 0, 0, 0, 0, 0]
  Call Extruder 0.00407
  MoveL (T8530) to (109.16, 105.38, 10.5) mm, rotated rx 180 ry 0 rz -180 deg; joints [0, 0, 0, 0, 0, 0]
  Call Extruder 0.00691
  MoveL (T8531) to (109.16, 105.19, 10.5) mm, rotated rx 180 ry 0 rz -180 deg; joints [0, 0, 0, 0, 0, 0]
  Call Extruder 0.0199
  MoveL (T8532) to (109.55, 104.79, 10.5) mm, rotated rx 180 ry 0 rz -180 deg; joints [0, 0, 0, 0, 0, 0]
  Call Extruder 0.02384
  MoveL (T8533) to (109.55, 104.12, 10.5) mm, rotated rx 180 ry 0 rz -180 deg; joints [0, 0, 0, 0, 0, 0]
  Call Extruder 0.0199
  MoveL (T8534) to (109.16, 104.52, 10.5) mm, rotated rx 180 ry 0 rz -180 deg; joints [0, 0, 0, 0, 0, 0]
  Call Extruder 0.02384
  MoveL (T8535) to (109.16, 103.84, 10.5) mm, rotated rx 180 ry 0 rz -180 deg; joints [0, 0, 0, 0, 0, 0]
  Call Extruder 0.00922
